RoboDK station: kr30 cnc 101019 2.rdk

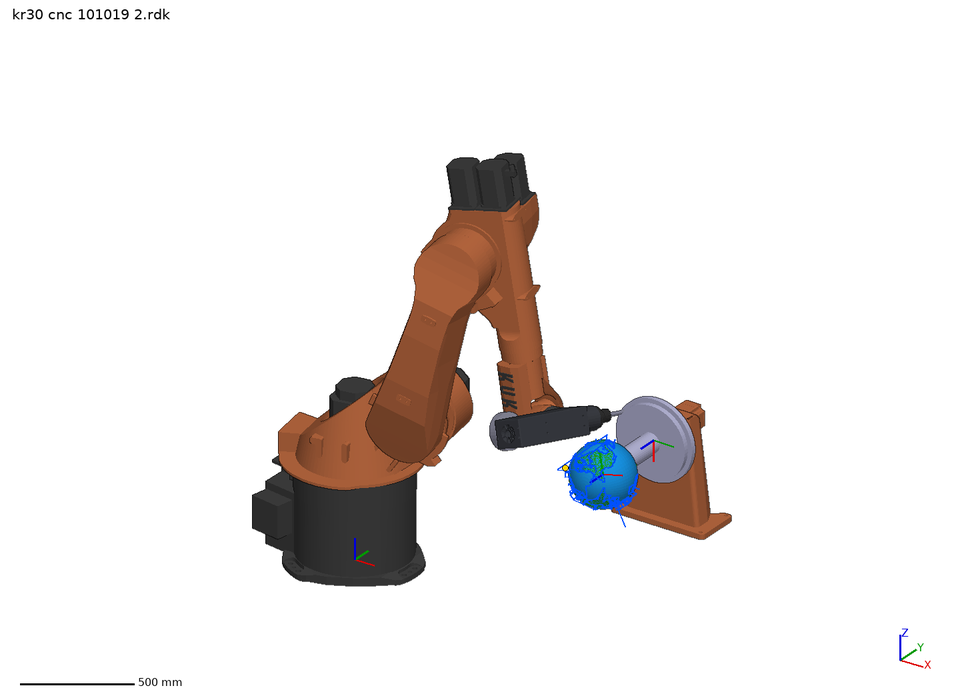
[picture v0: the station drawn from its stored meshes, robots at their saved joint values, targets as dots, program paths as lines]
Station kr30 cnc 101019 2. Poses are relative to the parent item; angles as X-Y-Z fixed-axis rotations.
  - frame KUKA KR 30 HA Base at (0, 0, 0) mm
    - robot KUKA KR 30 HA: 6 axes, payload 30 kg, reach 2033 mm, repeatability 0.05 mm, weight 665 kg
        modified DH rows (alpha deg, a mm, theta deg, d mm): 0, 0, 0, 815; -90, 350, 0, 0; 0, 850, -90, 0; -90, 145, 0, 820; 90, 0, 0, 0; -90, 0, 180, 170
        joint limits [-185, -135, -120, -350, -119, -350] to [185, 35, 158, 350, 119, 350]; home [0, -90, 90, 0, 0, 0]; saved at [-9.82, -73.833, 154.586, -18.357, -102.464, -76.723]
      - tool Spindle, TCP at (249.17, -0.03, 160.93) mm, rotated rx 0 ry 90 rz 0 deg, size 170 x 692.9 x 256 mm
  - frame KUKA KP1 MD250 Base at (1360.87, 339.35, 824.43) mm, rotated rx -93.1 ry 88.62 rz 178.42 deg
    - robot KUKA KP1 MD250: 1 axes, payload 250 kg
        modified DH rows (alpha deg, a mm, theta deg, d mm): 0, 0, 0, 0
        joint limits [-180] to [180]; home [0]; saved at [-257.733]
      - frame MillingEarth at (0, 0, 402.47) mm
        - object Earth at (0, 0, 0) mm, size 359.7 x 359.7 x 550 mm
  - machining project MillingEarth Settings: C:/Users/albert/Desktop/RoboDK/Deploy/RoboDK_vc2013x64/Library/Milling Earth (5axis).nc | rotZ(0) | rotX(0)*rotY(0) | rotZ(90)
  - program MillingEarth (2694 instructions, listed below)
  - program Prog2 (0 instructions, listed below)
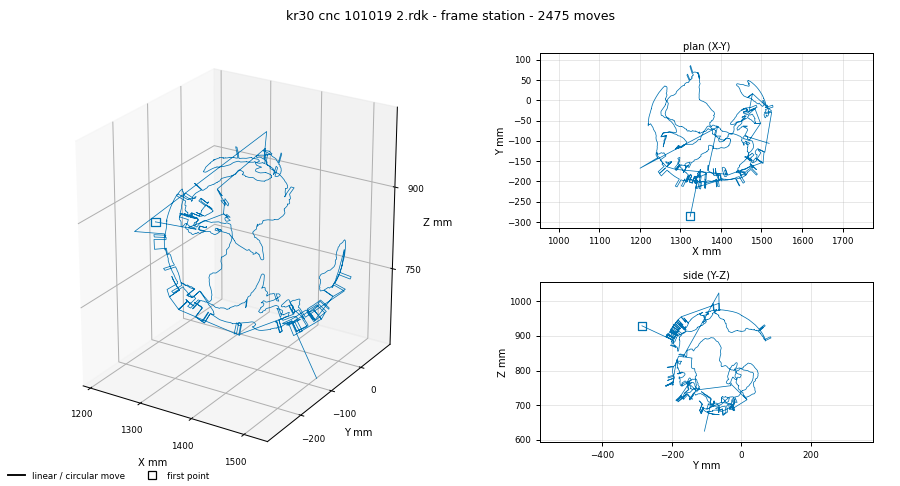
[picture p0: tool path of kr30 cnc 101019 2.rdk in frame station, 2475 of 2475 moves have a stored position in this frame; points joined in program order, loops and branches not executed]

--- program MillingEarth (robot KUKA KR 30 HA) ---
  Call onMillingEarth_Start
  Set Ref.: MillingEarth
  Set Tool: Spindle
  Show Spindle
  Set speed (16.7 mm/s)
  Call SetCLW
  Call SetRPM(70.0)
  Set speed (1000.0 mm/s)
  MoveJ 1 to (-32.4, 113.46, 221.55) mm, rotated rx -152.37 ry 0 rz -164.91 deg; joints [17.149, -48.365, 79.155, 0, 59.444, -43.7, -13.927]
  MoveL 2 to (-32.4, 113.46, 221.55) mm, rotated rx -152.37 ry 0 rz -164.91 deg; joints [17.149, -48.365, 79.155, 0, 59.444, -43.7, -13.926]
  Call onMillingEarth_Approach
  MoveL 3 to (-20.33, 68.69, 132.95) mm, rotated rx -152.37 ry 0 rz -164.91 deg; joints [14.531, -51.571, 85.433, 1.012, 59.444, -46.856, -17.119]
  Call onMillingEarth_PathStart
  MoveL 4 to (-20.33, 68.69, 132.95) mm, rotated rx -152.37 ry 0 rz -164.91 deg; joints [14.531, -51.571, 85.433, 1.012, 59.444, -46.856, -17.119]
  MoveL 5 to (-19.96, 69.22, 132.73) mm, rotated rx -152.2 ry 0 rz -165.3 deg; joints [14.503, -51.529, 85.357, 0.999, 59.444, -46.702, -16.7]
  Set speed (16.7 mm/s)
  MoveL 6 to (-22.33, 78.24, 150.42) mm, rotated rx -152.2 ry 0 rz -165.3 deg; joints [15.035, -50.886, 84.143, 0.841, 59.444, -46.082, -16.114]
  Set speed (1000.0 mm/s)
  MoveL 7 to (39.62, 97.38, 134.89) mm, rotated rx -142.85 ry 0 rz 157.38 deg; joints [13.369, -48.767, 80.092, 0.147, 59.444, -38.037, 23.226]
  Set speed (5.0 mm/s)
  MoveL 8 to (34.97, 86.23, 118.95) mm, rotated rx -142.85 ry 0 rz 157.38 deg; joints [12.91, -49.457, 81.504, 0.356, 59.444, -38.604, 22.481]
  Set speed (16.7 mm/s)
  MoveL 9 to (35.17, 86.21, 118.9) mm, rotated rx -142.83 ry 0 rz 157.26 deg; joints [12.906, -49.452, 81.493, 0.354, 59.444, -38.581, 22.605]
  MoveL 10 to (35.37, 86.18, 118.87) mm, rotated rx -142.83 ry 0 rz 157.26 deg; joints [12.904, -49.443, 81.493, 0.355, 59.439, -38.583, 22.602]
  MoveL 11 to (39.2, 85.43, 118.2) mm, rotated rx -142.42 ry 0 rz 154.93 deg; joints [12.831, -49.365, 81.337, 0.33, 59.439, -38.237, 25.012]
  MoveL 12 to (44.37, 96.48, 134.05) mm, rotated rx -142.42 ry 0 rz 154.93 deg; joints [13.286, -48.674, 79.917, 0.119, 59.439, -37.672, 25.764]
  Set speed (1000.0 mm/s)
  MoveL 13 to (45.45, 92.09, 136.75) mm, rotated rx -142.45 ry 0 rz 154.62 deg; joints [13.396, -48.674, 80.171, 0.201, 59.442, -37.638, 25.808]
  Set speed (5.0 mm/s)
  MoveL 14 to (40.23, 81.08, 120.9) mm, rotated rx -142.45 ry 0 rz 154.62 deg; joints [12.942, -49.369, 81.594, 0.41, 59.443, -38.201, 25.058]
  Set speed (16.7 mm/s)
  MoveL 15 to (37.93, 80.72, 121.87) mm, rotated rx -143.08 ry 0 rz 155.86 deg; joints [13.052, -49.49, 81.836, 0.45, 59.443, -38.738, 23.689]
  MoveL 16 to (37.59, 80.7, 121.99) mm, rotated rx -143.15 ry 0 rz 156.04 deg; joints [13.065, -49.505, 81.863, 0.454, 59.443, -38.795, 23.499]
  MoveL 17 to (35.64, 80.36, 122.8) mm, rotated rx -143.67 ry 0 rz 157.12 deg; joints [13.157, -49.609, 82.069, 0.489, 59.443, -39.247, 22.314]
  MoveL 18 to (35.2, 80.32, 122.95) mm, rotated rx -143.67 ry 0 rz 157.12 deg; joints [13.164, -49.63, 82.075, 0.489, 59.457, -39.24, 22.314]
  MoveL 19 to (34.17, 80.49, 123.13) mm, rotated rx -143.67 ry 0 rz 157.12 deg; joints [13.173, -49.678, 82.075, 0.482, 59.484, -39.227, 22.337]
  MoveL 20 to (33.97, 80.56, 123.14) mm, rotated rx -143.68 ry 0 rz 157.26 deg; joints [13.174, -49.679, 82.077, 0.483, 59.484, -39.233, 22.196]
  MoveL 21 to (33.46, 80.79, 123.13) mm, rotated rx -143.68 ry 0 rz 157.26 deg; joints [13.175, -49.708, 82.074, 0.473, 59.484, -39.227, 22.228]
  MoveL 22 to (32.55, 81.6, 122.84) mm, rotated rx -143.68 ry 0 rz 157.26 deg; joints [13.166, -49.754, 82.043, 0.449, 59.484, -39.223, 22.308]
  MoveL 23 to (31.58, 82.93, 122.2) mm, rotated rx -143.26 ry 0 rz 158.18 deg; joints [13.092, -49.671, 81.88, 0.422, 59.484, -38.865, 21.471]
  MoveL 24 to (31.06, 83.97, 121.62) mm, rotated rx -143.25 ry 0 rz 158.2 deg; joints [13.068, -49.685, 81.82, 0.399, 59.484, -38.861, 21.523]
  MoveL 25 to (31.07, 84.77, 121.06) mm, rotated rx -143.23 ry 0 rz 158.22 deg; joints [13.044, -49.671, 81.765, 0.386, 59.483, -38.866, 21.548]
  MoveL 26 to (31.31, 85.29, 120.63) mm, rotated rx -143.22 ry 0 rz 158.24 deg; joints [13.025, -49.647, 81.723, 0.38, 59.483, -38.874, 21.553]
  MoveL 27 to (31.95, 85.85, 120.07) mm, rotated rx -143.21 ry 0 rz 158.26 deg; joints [12.999, -49.604, 81.676, 0.373, 59.469, -38.883, 21.553]
  MoveL 28 to (32.84, 86.09, 119.65) mm, rotated rx -143.2 ry 0 rz 158.27 deg; joints [12.98, -49.563, 81.657, 0.367, 59.428, -38.887, 21.553]
  MoveL 29 to (34.47, 86.24, 119.09) mm, rotated rx -142.85 ry 0 rz 157.38 deg; joints [12.918, -49.496, 81.523, 0.345, 59.428, -38.591, 22.517]
  MoveL 30 to (39.12, 97.38, 135.03) mm, rotated rx -142.85 ry 0 rz 157.38 deg; joints [13.377, -48.806, 80.112, 0.137, 59.428, -38.024, 23.262]
  Set speed (1000.0 mm/s)
  MoveL 31 to (36.17, 117.37, 119.01) mm, rotated rx -134.2 ry 0 rz 164.03 deg; joints [11.734, -47.132, 76.943, -0.298, 59.428, -30.795, 18.15]
  Set speed (5.0 mm/s)
  MoveL 32 to (32.22, 103.58, 105.07) mm, rotated rx -134.2 ry 0 rz 164.03 deg; joints [11.348, -47.847, 78.519, -0.063, 59.428, -31.299, 17.264]
  Set speed (16.7 mm/s)
  MoveL 33 to (31.89, 100.84, 107.81) mm, rotated rx -135.66 ry 0 rz 163.8 deg; joints [11.629, -48.075, 79.013, 0.01, 59.428, -32.518, 17.226]
  MoveL 34 to (35.79, 114.26, 122.11) mm, rotated rx -135.66 ry 0 rz 163.8 deg; joints [12.027, -47.363, 77.462, -0.222, 59.428, -32.002, 18.089]
  Set speed (1000.0 mm/s)
  MoveL 35 to (30.39, 115.24, 122.66) mm, rotated rx -135.75 ry 0 rz 164.03 deg; joints [12.066, -47.602, 77.462, -0.26, 59.533, -32.027, 17.992]
  Set speed (5.0 mm/s)
  MoveL 36 to (26.55, 101.82, 108.33) mm, rotated rx -135.75 ry 0 rz 164.03 deg; joints [11.666, -48.313, 79.006, -0.028, 59.533, -32.543, 17.134]
  Set speed (16.7 mm/s)
  MoveL 37 to (26.92, 104.59, 105.56) mm, rotated rx -134.26 ry 0 rz 164.25 deg; joints [11.381, -48.081, 78.504, -0.101, 59.533, -31.302, 17.192]
  MoveL 38 to (30.8, 118.38, 119.52) mm, rotated rx -134.26 ry 0 rz 164.25 deg; joints [11.768, -47.367, 76.934, -0.336, 59.533, -30.798, 18.073]
  Set speed (1000.0 mm/s)
  MoveL 39 to (18.54, 129.47, 110.19) mm, rotated rx -130.91 ry 0 rz 171.49 deg; joints [11.006, -46.736, 75.687, -0.48, 59.533, -28.141, 11.458]
  Set speed (5.0 mm/s)
  MoveL 40 to (16.3, 114.52, 97.09) mm, rotated rx -130.91 ry 0 rz 171.49 deg; joints [10.647, -47.452, 77.314, -0.24, 59.533, -28.616, 10.522]
  Set speed (16.7 mm/s)
  MoveL 41 to (17.17, 114.58, 96.87) mm, rotated rx -130.8 ry 0 rz 171.07 deg; joints [10.625, -47.437, 77.281, -0.245, 59.533, -28.526, 10.961]
  MoveL 42 to (17.11, 114.6, 96.86) mm, rotated rx -128.95 ry 0 rz 171.63 deg; joints [10.392, -47.226, 76.933, -0.275, 59.533, -26.899, 10.541]
  MoveL 43 to (16.23, 114.67, 96.93) mm, rotated rx -128.98 ry 0 rz 172.06 deg; joints [10.399, -47.23, 76.942, -0.273, 59.535, -26.926, 10.101]
  MoveL 44 to (18.38, 130.06, 109.51) mm, rotated rx -128.98 ry 0 rz 172.06 deg; joints [10.74, -46.507, 75.283, -0.515, 59.535, -26.468, 11.062]
  Set speed (1000.0 mm/s)
  MoveL 45 to (51.72, 163.01, 1.41) mm, rotated rx -91.23 ry 0 rz 162.75 deg; joints [1.995, -46.507, 71.751, -0.724, 56.15, 2.635, 27.263]
  Set speed (5.0 mm/s)
  MoveL 46 to (45.79, 143.91, 0.98) mm, rotated rx -91.23 ry 0 rz 162.75 deg; joints [2.004, -47.144, 73.595, -0.637, 56.154, 2.607, 26.05]
  Set speed (16.7 mm/s)
  MoveL 47 to (46.25, 143.76, 1.2) mm, rotated rx -91.32 ry 0 rz 162.56 deg; joints [2.023, -47.144, 73.594, -0.64, 56.152, 2.544, 26.237]
  MoveL 48 to (46.82, 143.57, 1.59) mm, rotated rx -91.32 ry 0 rz 162.56 deg; joints [2.036, -47.115, 73.594, -0.641, 56.139, 2.557, 26.221]
  MoveL 49 to (49.93, 142.45, 4.46) mm, rotated rx -92.41 ry 0 rz 161.31 deg; joints [2.289, -47.115, 73.581, -0.683, 56.12, 1.741, 27.508]
  MoveL 50 to (49.93, 142.46, 4.45) mm, rotated rx -92.58 ry 0 rz 161.02 deg; joints [2.313, -47.154, 73.581, -0.689, 56.13, 1.6, 27.828]
  MoveL 51 to (53.02, 141.29, 5.69) mm, rotated rx -93.05 ry 0 rz 159.77 deg; joints [2.422, -47.154, 73.578, -0.707, 56.124, 1.249, 29.091]
  MoveL 52 to (53.52, 141.09, 5.97) mm, rotated rx -93.05 ry 0 rz 159.77 deg; joints [2.431, -47.127, 73.578, -0.707, 56.114, 1.258, 29.075]
  MoveL 53 to (54.32, 140.74, 7.02) mm, rotated rx -93.05 ry 0 rz 159.77 deg; joints [2.465, -47.084, 73.578, -0.71, 56.096, 1.295, 29.051]
  MoveL 54 to (54.41, 140.69, 7.24) mm, rotated rx -93.13 ry 0 rz 159.73 deg; joints [2.484, -47.084, 73.578, -0.714, 56.095, 1.233, 29.088]
  MoveL 55 to (54.58, 140.57, 8.16) mm, rotated rx -93.13 ry 0 rz 159.73 deg; joints [2.515, -47.074, 73.578, -0.718, 56.089, 1.266, 29.085]
  MoveL 56 to (54.59, 140.48, 9.51) mm, rotated rx -93.64 ry 0 rz 159.71 deg; joints [2.634, -47.074, 73.577, -0.737, 56.085, 0.883, 29.106]
  MoveL 57 to (54.58, 140.49, 9.48) mm, rotated rx -94.31 ry 0 rz 159.4 deg; joints [2.73, -47.115, 73.577, -0.754, 56.097, 0.318, 29.449]
  MoveL 58 to (58.8, 138.43, 13.63) mm, rotated rx -95.89 ry 0 rz 157.62 deg; joints [3.095, -47.113, 73.586, -0.811, 56.097, -0.865, 31.221]
  MoveL 59 to (58.75, 138.46, 13.59) mm, rotated rx -96.1 ry 0 rz 157.16 deg; joints [3.126, -47.174, 73.586, -0.819, 56.123, -1.045, 31.719]
  MoveL 60 to (63.19, 136.41, 14.38) mm, rotated rx -96.4 ry 0 rz 155.3 deg; joints [3.195, -47.174, 73.59, -0.829, 56.123, -1.269, 33.577]
  MoveL 61 to (63.44, 136.29, 14.44) mm, rotated rx -96.4 ry 0 rz 155.3 deg; joints [3.197, -47.16, 73.59, -0.829, 56.119, -1.268, 33.568]
  MoveL 62 to (63.67, 136.17, 14.51) mm, rotated rx -96.43 ry 0 rz 155.2 deg; joints [3.203, -47.16, 73.59, -0.83, 56.119, -1.288, 33.667]
  MoveL 63 to (65.41, 135.28, 15.07) mm, rotated rx -96.66 ry 0 rz 154.35 deg; joints [3.257, -47.171, 73.59, -0.838, 56.13, -1.47, 34.516]
  MoveL 64 to (65.72, 135.13, 15.13) mm, rotated rx -96.69 ry 0 rz 154.22 deg; joints [3.261, -47.171, 73.591, -0.839, 56.13, -1.485, 34.646]
  MoveL 65 to (68.28, 133.79, 15.64) mm, rotated rx -96.88 ry 0 rz 153.13 deg; joints [3.306, -47.169, 73.594, -0.845, 56.13, -1.63, 35.729]
  MoveL 66 to (68.86, 133.47, 15.86) mm, rotated rx -96.88 ry 0 rz 153.13 deg; joints [3.313, -47.135, 73.594, -0.844, 56.119, -1.624, 35.707]
  MoveL 67 to (69.74, 132.95, 16.36) mm, rotated rx -97.07 ry 0 rz 152.75 deg; joints [3.357, -47.133, 73.595, -0.85, 56.125, -1.766, 36.083]
  MoveL 68 to (69.89, 132.86, 16.45) mm, rotated rx -97.07 ry 0 rz 152.75 deg; joints [3.36, -47.124, 73.595, -0.85, 56.122, -1.763, 36.077]
  MoveL 69 to (76.53, 128.45, 21.19) mm, rotated rx -98.88 ry 0 rz 149.71 deg; joints [3.778, -47.124, 73.638, -0.908, 56.143, -3.127, 39.054]
  MoveL 70 to (76.49, 128.48, 21.19) mm, rotated rx -98.98 ry 0 rz 148.97 deg; joints [3.794, -47.219, 73.638, -0.916, 56.183, -3.206, 39.853]
  MoveL 71 to (80.12, 126.44, 20.02) mm, rotated rx -98.53 ry 0 rz 147.38 deg; joints [3.69, -47.219, 73.625, -0.902, 56.176, -2.867, 41.464]
  MoveL 72 to (80.83, 126, 19.93) mm, rotated rx -98.53 ry 0 rz 147.38 deg; joints [3.686, -47.179, 73.625, -0.899, 56.16, -2.872, 41.439]
  MoveL 73 to (81.28, 125.71, 19.96) mm, rotated rx -98.54 ry 0 rz 147.17 deg; joints [3.689, -47.179, 73.625, -0.9, 56.16, -2.881, 41.642]
  MoveL 74 to (81.75, 125.39, 20.06) mm, rotated rx -98.54 ry 0 rz 147.17 deg; joints [3.692, -47.15, 73.625, -0.898, 56.15, -2.879, 41.623]
  MoveL 75 to (86.58, 121.8, 21.83) mm, rotated rx -99.22 ry 0 rz 144.87 deg; joints [3.849, -47.15, 73.644, -0.919, 56.161, -3.392, 43.899]
  MoveL 76 to (87.18, 121.32, 22.1) mm, rotated rx -99.31 ry 0 rz 144.62 deg; joints [3.87, -47.145, 73.647, -0.921, 56.161, -3.457, 44.142]
  MoveL 77 to (91.51, 117.76, 23.78) mm, rotated rx -99.97 ry 0 rz 142.43 deg; joints [4.02, -47.145, 73.663, -0.94, 56.184, -3.955, 46.29]
  MoveL 78 to (91.73, 117.56, 23.89) mm, rotated rx -99.97 ry 0 rz 142.43 deg; joints [4.023, -47.13, 73.664, -0.939, 56.179, -3.952, 46.28]
  MoveL 79 to (92.05, 117.28, 24.08) mm, rotated rx -100.04 ry 0 rz 142.27 deg; joints [4.04, -47.13, 73.667, -0.942, 56.18, -4.006, 46.437]
  MoveL 80 to (92.22, 117.12, 24.19) mm, rotated rx -100.04 ry 0 rz 142.27 deg; joints [4.044, -47.118, 73.666, -0.941, 56.178, -4.003, 46.428]
  MoveL 81 to (94.43, 114.96, 25.97) mm, rotated rx -100.72 ry 0 rz 141.09 deg; joints [4.2, -47.118, 73.692, -0.96, 56.194, -4.518, 47.571]
  MoveL 82 to (96.38, 113.21, 26.49) mm, rotated rx -101.03 ry 0 rz 139.79 deg; joints [4.263, -47.144, 73.692, -0.968, 56.231, -4.763, 48.857]
  MoveL 83 to (96.7, 112.9, 26.63) mm, rotated rx -101.03 ry 0 rz 139.79 deg; joints [4.267, -47.121, 73.692, -0.967, 56.225, -4.759, 48.84]
  MoveL 84 to (96.94, 112.66, 26.77) mm, rotated rx -101.08 ry 0 rz 139.66 deg; joints [4.279, -47.121, 73.694, -0.968, 56.226, -4.8, 48.967]
  MoveL 85 to (97.15, 112.45, 26.91) mm, rotated rx -101.08 ry 0 rz 139.66 deg; joints [4.284, -47.105, 73.694, -0.967, 56.223, -4.796, 48.955]
  MoveL 86 to (99.43, 109.95, 28.85) mm, rotated rx -101.83 ry 0 rz 138.37 deg; joints [4.455, -47.105, 73.726, -0.986, 56.245, -5.361, 50.196]
  MoveL 87 to (99.68, 109.66, 29.07) mm, rotated rx -101.92 ry 0 rz 138.21 deg; joints [4.475, -47.105, 73.73, -0.988, 56.249, -5.428, 50.343]
  MoveL 88 to (100.05, 109.21, 29.52) mm, rotated rx -101.92 ry 0 rz 138.21 deg; joints [4.489, -47.074, 73.73, -0.987, 56.246, -5.415, 50.314]
  MoveL 89 to (101.45, 107.18, 32.04) mm, rotated rx -102.89 ry 0 rz 137.28 deg; joints [4.712, -47.075, 73.778, -1.01, 56.278, -6.156, 51.167]
  MoveL 90 to (101.64, 106.86, 32.53) mm, rotated rx -102.89 ry 0 rz 137.28 deg; joints [4.728, -47.055, 73.779, -1.009, 56.278, -6.14, 51.146]
  MoveL 91 to (101.66, 106.43, 33.85) mm, rotated rx -102.89 ry 0 rz 137.28 deg; joints [4.772, -47.041, 73.791, -1.013, 56.278, -6.094, 51.121]
  MoveL 92 to (101.59, 106.39, 34.17) mm, rotated rx -103.02 ry 0 rz 137.29 deg; joints [4.8, -47.041, 73.798, -1.015, 56.283, -6.188, 51.102]
  MoveL 93 to (101.26, 106.41, 35.09) mm, rotated rx -103.02 ry 0 rz 137.29 deg; joints [4.831, -47.047, 73.798, -1.017, 56.305, -6.156, 51.086]
  MoveL 94 to (100.18, 106.74, 37.1) mm, rotated rx -103.8 ry 0 rz 137.69 deg; joints [5.01, -47.047, 73.842, -1.033, 56.338, -6.756, 50.61]
  MoveL 95 to (100.18, 106.75, 37.07) mm, rotated rx -104.74 ry 0 rz 137.63 deg; joints [5.141, -47.047, 73.868, -1.042, 56.38, -7.555, 50.606]
  MoveL 96 to (101.87, 103.05, 42.54) mm, rotated rx -107.02 ry 0 rz 136.04 deg; joints [5.645, -47.047, 74.005, -1.07, 56.529, -9.322, 51.922]
  MoveL 97 to (102.05, 102.73, 42.88) mm, rotated rx -107.16 ry 0 rz 135.9 deg; joints [5.676, -47.047, 74.015, -1.072, 56.537, -9.425, 52.043]
  MoveL 98 to (104.05, 99.2, 46.26) mm, rotated rx -108.54 ry 0 rz 134.31 deg; joints [5.982, -47.047, 74.116, -1.081, 56.635, -10.493, 53.437]
  MoveL 99 to (104.28, 98.54, 47.15) mm, rotated rx -108.59 ry 0 rz 134.31 deg; joints [6.018, -47.015, 74.131, -1.079, 56.635, -10.506, 53.387]
  MoveL 100 to (104.13, 98.18, 48.22) mm, rotated rx -108.63 ry 0 rz 134.31 deg; joints [6.06, -47.013, 74.153, -1.081, 56.635, -10.509, 53.359]
  MoveL 101 to (103.98, 98.01, 48.88) mm, rotated rx -108.9 ry 0 rz 134.31 deg; joints [6.119, -47.013, 74.176, -1.082, 56.654, -10.716, 53.322]
  MoveL 102 to (103.97, 98.04, 48.86) mm, rotated rx -109.5 ry 0 rz 134.07 deg; joints [6.202, -47.014, 74.176, -1.077, 56.743, -11.239, 53.472]
  MoveL 103 to (104.32, 97.19, 49.77) mm, rotated rx -109.87 ry 0 rz 133.73 deg; joints [6.284, -47.014, 74.209, -1.077, 56.771, -11.525, 53.754]
  MoveL 104 to (104.27, 97.22, 49.84) mm, rotated rx -109.04 ry 0 rz 132.02 deg; joints [6.179, -47.246, 74.182, -1.106, 56.771, -10.79, 55.725]
  MoveL 105 to (104.53, 98.86, 45.91) mm, rotated rx -107.47 ry 0 rz 132.44 deg; joints [5.826, -47.246, 74.054, -1.096, 56.663, -9.572, 55.539]
  MoveL 106 to (104.48, 99.07, 45.58) mm, rotated rx -107.19 ry 0 rz 132.57 deg; joints [5.777, -47.246, 74.044, -1.095, 56.636, -9.348, 55.449]
  MoveL 107 to (104.22, 100.62, 42.67) mm, rotated rx -106.04 ry 0 rz 133.09 deg; joints [5.517, -47.246, 73.959, -1.082, 56.568, -8.458, 55.076]
  MoveL 108 to (118.26, 113.75, 48.19) mm, rotated rx -106.04 ry 0 rz 133.09 deg; joints [5.653, -46.589, 72.136, -1.276, 56.567, -8.236, 56.255]
  Set speed (1000.0 mm/s)
  MoveL 109 to (121.75, 111.27, 45.2) mm, rotated rx -106.02 ry 0 rz 132.91 deg; joints [5.547, -46.443, 72.136, -1.261, 56.421, -8.333, 56.435]
  Set speed (5.0 mm/s)
  MoveL 110 to (107.67, 98.18, 39.68) mm, rotated rx -106.02 ry 0 rz 132.91 deg; joints [5.411, -47.099, 73.963, -1.068, 56.421, -8.555, 55.251]
  Set speed (16.7 mm/s)
  MoveL 111 to (109.17, 95.75, 41.47) mm, rotated rx -106.73 ry 0 rz 131.8 deg; joints [5.57, -47.099, 74.013, -1.077, 56.46, -9.097, 56.269]
  MoveL 112 to (109.28, 95.57, 41.61) mm, rotated rx -106.78 ry 0 rz 131.72 deg; joints [5.582, -47.099, 74.017, -1.078, 56.463, -9.138, 56.345]
  MoveL 113 to (110.67, 92.99, 43.73) mm, rotated rx -107.58 ry 0 rz 130.65 deg; joints [5.765, -47.099, 74.085, -1.088, 56.497, -9.747, 57.313]
  MoveL 114 to (110.84, 92.61, 44.1) mm, rotated rx -107.58 ry 0 rz 130.65 deg; joints [5.777, -47.078, 74.087, -1.086, 56.497, -9.736, 57.289]
  MoveL 115 to (110.92, 91.99, 45.19) mm, rotated rx -107.58 ry 0 rz 130.65 deg; joints [5.813, -47.053, 74.101, -1.085, 56.497, -9.701, 57.251]
  MoveL 116 to (110.89, 91.91, 45.44) mm, rotated rx -107.68 ry 0 rz 130.63 deg; joints [5.835, -47.053, 74.109, -1.086, 56.504, -9.776, 57.255]
  MoveL 117 to (110.71, 91.74, 46.19) mm, rotated rx -107.68 ry 0 rz 130.63 deg; joints [5.86, -47.053, 74.118, -1.087, 56.51, -9.75, 57.24]
  MoveL 118 to (110.22, 91.6, 47.62) mm, rotated rx -108.25 ry 0 rz 130.72 deg; joints [5.989, -47.053, 74.165, -1.09, 56.548, -10.194, 57.07]
  MoveL 119 to (110.22, 91.62, 47.57) mm, rotated rx -109.14 ry 0 rz 130.3 deg; joints [6.11, -47.061, 74.165, -1.086, 56.679, -10.967, 57.364]
  MoveL 120 to (112.14, 87.75, 50.32) mm, rotated rx -110.24 ry 0 rz 128.62 deg; joints [6.355, -47.061, 74.261, -1.088, 56.761, -11.82, 58.874]
  MoveL 121 to (112.4, 86.84, 51.32) mm, rotated rx -110.24 ry 0 rz 128.62 deg; joints [6.388, -47.017, 74.274, -1.082, 56.761, -11.79, 58.816]
  MoveL 122 to (112.13, 86.41, 52.6) mm, rotated rx -110.24 ry 0 rz 128.62 deg; joints [6.431, -47.016, 74.3, -1.083, 56.761, -11.746, 58.79]
  MoveL 123 to (112.01, 86.37, 52.93) mm, rotated rx -110.38 ry 0 rz 128.64 deg; joints [6.461, -47.017, 74.313, -1.083, 56.77, -11.85, 58.747]
  MoveL 124 to (111.32, 86.54, 54.09) mm, rotated rx -110.38 ry 0 rz 128.64 deg; joints [6.5, -47.029, 74.313, -1.081, 56.82, -11.812, 58.709]
  MoveL 125 to (110.56, 86.95, 54.96) mm, rotated rx -110.73 ry 0 rz 128.96 deg; joints [6.579, -47.033, 74.352, -1.081, 56.843, -12.09, 58.33]
  MoveL 126 to (110.59, 86.95, 54.91) mm, rotated rx -111.91 ry 0 rz 128.97 deg; joints [6.74, -47.043, 74.434, -1.081, 56.887, -13.111, 58.207]
  MoveL 127 to (110.98, 85.3, 56.68) mm, rotated rx -112.64 ry 0 rz 128.35 deg; joints [6.9, -47.06, 74.524, -1.081, 56.923, -13.674, 58.722]
  MoveL 128 to (111.01, 84.82, 57.35) mm, rotated rx -112.64 ry 0 rz 128.35 deg; joints [6.922, -47.042, 74.537, -1.078, 56.923, -13.653, 58.691]
  MoveL 129 to (110.99, 84.64, 57.66) mm, rotated rx -112.76 ry 0 rz 128.3 deg; joints [6.95, -47.046, 74.554, -1.078, 56.929, -13.752, 58.721]
  MoveL 130 to (110.91, 84.43, 58.11) mm, rotated rx -112.76 ry 0 rz 128.3 deg; joints [6.965, -47.043, 74.565, -1.077, 56.929, -13.737, 58.708]
  MoveL 131 to (110.03, 83.05, 61.67) mm, rotated rx -114.23 ry 0 rz 128.08 deg; joints [7.289, -47.102, 74.782, -1.077, 56.976, -14.882, 58.727]
  MoveL 132 to (109.88, 82.87, 62.17) mm, rotated rx -114.4 ry 0 rz 128.06 deg; joints [7.328, -47.111, 74.811, -1.077, 56.98, -15.003, 58.718]
  MoveL 133 to (109.06, 81.95, 64.77) mm, rotated rx -115.48 ry 0 rz 127.97 deg; joints [7.566, -47.171, 74.996, -1.077, 56.996, -15.847, 58.674]
  MoveL 134 to (109.07, 81.98, 64.73) mm, rotated rx -116.1 ry 0 rz 127.61 deg; joints [7.65, -47.221, 75.046, -1.077, 57.042, -16.387, 58.982]
  MoveL 135 to (109.68, 79.86, 66.33) mm, rotated rx -116.77 ry 0 rz 126.75 deg; joints [7.796, -47.266, 75.171, -1.077, 57.044, -16.909, 59.764]
  MoveL 136 to (109.69, 79.87, 66.3) mm, rotated rx -116.91 ry 0 rz 126.48 deg; joints [7.815, -47.29, 75.173, -1.077, 57.075, -17.033, 60.026]
  MoveL 137 to (110.88, 77.27, 67.41) mm, rotated rx -117.38 ry 0 rz 125.3 deg; joints [7.916, -47.323, 75.264, -1.077, 57.075, -17.396, 61.148]
  MoveL 138 to (111.03, 76.87, 67.61) mm, rotated rx -117.38 ry 0 rz 125.3 deg; joints [7.922, -47.301, 75.267, -1.072, 57.075, -17.392, 61.123]
  MoveL 139 to (111.15, 76.07, 68.3) mm, rotated rx -117.38 ry 0 rz 125.3 deg; joints [7.945, -47.267, 75.284, -1.065, 57.075, -17.373, 61.072]
  MoveL 140 to (111.14, 75.85, 68.56) mm, rotated rx -117.49 ry 0 rz 125.23 deg; joints [7.969, -47.275, 75.306, -1.064, 57.075, -17.459, 61.131]
  MoveL 141 to (111.07, 75.48, 69.1) mm, rotated rx -117.49 ry 0 rz 125.23 deg; joints [7.987, -47.267, 75.322, -1.062, 57.075, -17.442, 61.107]
  MoveL 142 to (110.3, 73.8, 72.07) mm, rotated rx -118.76 ry 0 rz 124.83 deg; joints [8.263, -47.364, 75.582, -1.057, 57.075, -18.44, 61.346]
  MoveL 143 to (110.19, 73.63, 72.41) mm, rotated rx -118.76 ry 0 rz 124.83 deg; joints [8.275, -47.364, 75.593, -1.056, 57.076, -18.429, 61.335]
  MoveL 144 to (110.02, 73.45, 72.86) mm, rotated rx -118.95 ry 0 rz 124.8 deg; joints [8.317, -47.379, 75.634, -1.055, 57.076, -18.581, 61.334]
  MoveL 145 to (109.94, 73.37, 73.05) mm, rotated rx -118.95 ry 0 rz 124.8 deg; joints [8.323, -47.38, 75.64, -1.054, 57.078, -18.575, 61.327]
  MoveL 146 to (108.02, 71.92, 77.24) mm, rotated rx -120.78 ry 0 rz 124.76 deg; joints [8.716, -47.532, 76.041, -1.04, 57.078, -20.017, 61.124]
  MoveL 147 to (107.85, 71.77, 77.62) mm, rotated rx -120.99 ry 0 rz 124.74 deg; joints [8.757, -47.549, 76.084, -1.038, 57.078, -20.182, 61.112]
  MoveL 148 to (105.63, 70.25, 81.94) mm, rotated rx -122.86 ry 0 rz 124.76 deg; joints [9.159, -47.722, 76.531, -1.015, 57.078, -21.661, 60.826]
  MoveL 149 to (104.84, 70.16, 83.03) mm, rotated rx -122.86 ry 0 rz 124.76 deg; joints [9.198, -47.757, 76.574, -1.015, 57.085, -21.621, 60.81]
  MoveL 150 to (104.53, 70.23, 83.36) mm, rotated rx -123.01 ry 0 rz 124.87 deg; joints [9.229, -47.771, 76.61, -1.013, 57.085, -21.738, 60.68]
  MoveL 151 to (104.24, 70.33, 83.64) mm, rotated rx -123.01 ry 0 rz 124.87 deg; joints [9.24, -47.785, 76.618, -1.013, 57.094, -21.728, 60.677]
  MoveL 152 to (101.64, 71.39, 85.9) mm, rotated rx -124.05 ry 0 rz 125.95 deg; joints [9.458, -47.887, 76.878, -0.995, 57.094, -22.56, 59.432]
  MoveL 153 to (101.65, 71.39, 85.9) mm, rotated rx -124.25 ry 0 rz 126.11 deg; joints [9.483, -47.88, 76.907, -0.989, 57.095, -22.736, 59.237]
  MoveL 154 to (99.95, 71.26, 87.98) mm, rotated rx -125.31 ry 0 rz 126.59 deg; joints [9.696, -47.979, 77.172, -0.968, 57.095, -23.594, 58.597]
  MoveL 155 to (99.56, 71.29, 88.39) mm, rotated rx -125.31 ry 0 rz 126.59 deg; joints [9.712, -47.997, 77.189, -0.968, 57.102, -23.579, 58.592]
  MoveL 156 to (99.1, 71.39, 88.83) mm, rotated rx -125.52 ry 0 rz 126.75 deg; joints [9.755, -48.019, 77.243, -0.964, 57.102, -23.745, 58.394]
  MoveL 157 to (98.75, 71.49, 89.13) mm, rotated rx -125.52 ry 0 rz 126.75 deg; joints [9.766, -48.036, 77.253, -0.963, 57.112, -23.734, 58.39]
  MoveL 158 to (93.79, 73.31, 92.93) mm, rotated rx -127.33 ry 0 rz 128.89 deg; joints [10.139, -48.235, 77.746, -0.921, 57.112, -25.196, 55.958]
  MoveL 159 to (93.53, 73.39, 93.13) mm, rotated rx -127.55 ry 0 rz 129.12 deg; joints [10.174, -48.241, 77.794, -0.913, 57.112, -25.386, 55.683]
  MoveL 160 to (88.83, 73.91, 97.23) mm, rotated rx -129.57 ry 0 rz 130.81 deg; joints [10.582, -48.48, 78.372, -0.857, 57.112, -27.019, 53.658]
  MoveL 161 to (88.79, 73.91, 97.27) mm, rotated rx -129.72 ry 0 rz 130.91 deg; joints [10.603, -48.482, 78.402, -0.851, 57.112, -27.157, 53.526]
  MoveL 162 to (87.4, 73.49, 98.82) mm, rotated rx -130.61 ry 0 rz 131.26 deg; joints [10.771, -48.583, 78.654, -0.823, 57.112, -27.886, 53.025]
  MoveL 163 to (87.43, 73.5, 98.79) mm, rotated rx -131.37 ry 0 rz 131.12 deg; joints [10.865, -48.659, 78.796, -0.811, 57.112, -28.556, 53.097]
  MoveL 164 to (87.12, 70.77, 101.04) mm, rotated rx -132.5 ry 0 rz 130.18 deg; joints [11.09, -48.808, 79.146, -0.771, 57.112, -29.482, 53.837]
  MoveL 165 to (86.99, 70.33, 101.46) mm, rotated rx -132.5 ry 0 rz 130.18 deg; joints [11.105, -48.805, 79.17, -0.765, 57.112, -29.47, 53.809]
  MoveL 166 to (86.3, 69.7, 102.47) mm, rotated rx -132.5 ry 0 rz 130.18 deg; joints [11.144, -48.83, 79.232, -0.757, 57.112, -29.435, 53.771]
  MoveL 167 to (86.12, 69.64, 102.67) mm, rotated rx -132.6 ry 0 rz 130.21 deg; joints [11.164, -48.844, 79.264, -0.753, 57.112, -29.52, 53.716]
  MoveL 168 to (85.06, 69.65, 103.54) mm, rotated rx -132.6 ry 0 rz 130.21 deg; joints [11.199, -48.898, 79.313, -0.753, 57.126, -29.485, 53.71]
  MoveL 169 to (83.74, 70.04, 104.35) mm, rotated rx -133.03 ry 0 rz 130.82 deg; joints [11.283, -48.957, 79.449, -0.737, 57.126, -29.838, 53.023]
  MoveL 170 to (83.76, 70.05, 104.32) mm, rotated rx -133.57 ry 0 rz 131.2 deg; joints [11.346, -48.963, 79.554, -0.713, 57.126, -30.328, 52.536]
  MoveL 171 to (82.94, 69.61, 105.27) mm, rotated rx -134.23 ry 0 rz 131.33 deg; joints [11.463, -49.047, 79.748, -0.688, 57.126, -30.883, 52.304]
  MoveL 172 to (82.78, 69.45, 105.51) mm, rotated rx -134.36 ry 0 rz 131.32 deg; joints [11.487, -49.065, 79.789, -0.683, 57.126, -30.987, 52.286]
  MoveL 173 to (81.07, 67.48, 108.08) mm, rotated rx -135.8 ry 0 rz 131.12 deg; joints [11.761, -49.275, 80.26, -0.623, 57.126, -32.186, 52.217]
  MoveL 174 to (91.57, 76.65, 122.42) mm, rotated rx -135.8 ry 0 rz 131.12 deg; joints [12.165, -48.59, 78.742, -0.882, 57.126, -31.652, 53.08]
  Set speed (1000.0 mm/s)
  MoveL 175 to (90.79, 72.41, 125.54) mm, rotated rx -137.12 ry 0 rz 129.8 deg; joints [12.444, -48.808, 79.243, -0.815, 57.126, -32.724, 54.119]
  Set speed (5.0 mm/s)
  MoveL 176 to (80.33, 63.7, 110.89) mm, rotated rx -137.12 ry 0 rz 129.8 deg; joints [12.029, -49.492, 80.739, -0.559, 57.126, -33.269, 53.277]
  Set speed (16.7 mm/s)
  MoveL 177 to (78.53, 62.71, 112.72) mm, rotated rx -138.15 ry 0 rz 130.02 deg; joints [12.224, -49.657, 81.101, -0.509, 57.126, -34.137, 52.852]
  MoveL 178 to (77.97, 61.99, 113.51) mm, rotated rx -138.89 ry 0 rz 129.9 deg; joints [12.342, -49.76, 81.323, -0.477, 57.126, -34.769, 52.845]
  MoveL 179 to (77.39, 61.55, 114.14) mm, rotated rx -138.89 ry 0 rz 129.9 deg; joints [12.368, -49.785, 81.372, -0.471, 57.126, -34.746, 52.82]
  MoveL 180 to (77.25, 61.49, 114.27) mm, rotated rx -138.96 ry 0 rz 129.93 deg; joints [12.382, -49.798, 81.399, -0.467, 57.126, -34.81, 52.778]
  MoveL 181 to (76.96, 61.41, 114.51) mm, rotated rx -138.96 ry 0 rz 129.93 deg; joints [12.392, -49.812, 81.418, -0.466, 57.126, -34.8, 52.774]
  MoveL 182 to (76.39, 61.28, 114.96) mm, rotated rx -139.22 ry 0 rz 130.09 deg; joints [12.44, -49.856, 81.512, -0.453, 57.126, -35.022, 52.56]
  MoveL 183 to (76.36, 61.31, 114.96) mm, rotated rx -140.09 ry 0 rz 130 deg; joints [12.54, -49.958, 81.706, -0.428, 57.126, -35.796, 52.564]
  MoveL 184 to (75.89, 58.95, 116.5) mm, rotated rx -140.99 ry 0 rz 129.11 deg; joints [12.706, -50.113, 82.037, -0.379, 57.126, -36.557, 53.27]
  MoveL 185 to (75.88, 58.99, 116.48) mm, rotated rx -141.42 ry 0 rz 128.03 deg; joints [12.757, -50.233, 82.107, -0.379, 57.178, -36.935, 54.349]
  MoveL 186 to (78.23, 55.19, 116.8) mm, rotated rx -141.6 ry 0 rz 125.37 deg; joints [12.791, -50.266, 82.176, -0.369, 57.178, -37.092, 56.972]
  MoveL 187 to (78.45, 54.73, 116.87) mm, rotated rx -141.6 ry 0 rz 125.37 deg; joints [12.792, -50.241, 82.182, -0.36, 57.178, -37.096, 56.941]
  MoveL 188 to (78.6, 54.34, 116.95) mm, rotated rx -141.65 ry 0 rz 125.13 deg; joints [12.801, -50.25, 82.2, -0.357, 57.178, -37.137, 57.173]
  MoveL 189 to (78.73, 53.86, 117.08) mm, rotated rx -141.65 ry 0 rz 125.13 deg; joints [12.805, -50.23, 82.211, -0.347, 57.179, -37.138, 57.14]
  MoveL 190 to (79.04, 52.14, 117.64) mm, rotated rx -141.99 ry 0 rz 124.18 deg; joints [12.867, -50.29, 82.338, -0.328, 57.179, -37.428, 58.021]
  MoveL 191 to (79, 52.2, 117.64) mm, rotated rx -141.9 ry 0 rz 122.48 deg; joints [12.865, -50.435, 82.318, -0.379, 57.178, -37.307, 59.893]
  MoveL 192 to (80.03, 51.74, 117.15) mm, rotated rx -141.6 ry 0 rz 121.92 deg; joints [12.811, -50.383, 82.208, -0.395, 57.178, -37.058, 60.512]
  MoveL 193 to (80.55, 51.42, 116.94) mm, rotated rx -141.6 ry 0 rz 121.92 deg; joints [12.802, -50.354, 82.199, -0.395, 57.158, -37.068, 60.512]
  MoveL 194 to (80.84, 51.2, 116.84) mm, rotated rx -141.54 ry 0 rz 121.71 deg; joints [12.791, -50.343, 82.177, -0.398, 57.158, -37.018, 60.727]
  MoveL 195 to (81.31, 50.73, 116.71) mm, rotated rx -141.54 ry 0 rz 121.71 deg; joints [12.785, -50.314, 82.177, -0.396, 57.136, -37.025, 60.719]
  MoveL 196 to (83.31, 48.21, 116.37) mm, rotated rx -141.34 ry 0 rz 119.81 deg; joints [12.748, -50.279, 82.103, -0.407, 57.136, -36.855, 62.663]
  MoveL 197 to (83.12, 48.42, 116.42) mm, rotated rx -141.33 ry 0 rz 119.71 deg; joints [12.75, -50.301, 82.103, -0.413, 57.139, -36.836, 62.779]
  MoveL 198 to (83.31, 48.23, 116.36) mm, rotated rx -141.29 ry 0 rz 119.56 deg; joints [12.744, -50.296, 82.091, -0.415, 57.139, -36.808, 62.936]
  MoveL 199 to (85.09, 46.58, 115.75) mm, rotated rx -140.91 ry 0 rz 118.12 deg; joints [12.675, -50.237, 81.952, -0.437, 57.139, -36.48, 64.46]
  MoveL 200 to (85.39, 46.24, 115.66) mm, rotated rx -140.91 ry 0 rz 118.12 deg; joints [12.671, -50.217, 81.952, -0.436, 57.123, -36.485, 64.455]
  MoveL 201 to (85.89, 45.32, 115.66) mm, rotated rx -140.91 ry 0 rz 118.12 deg; joints [12.668, -50.161, 81.952, -0.42, 57.121, -36.496, 64.4]
  MoveL 202 to (85.97, 45.07, 115.69) mm, rotated rx -140.93 ry 0 rz 117.97 deg; joints [12.671, -50.164, 81.96, -0.419, 57.121, -36.513, 64.548]
  MoveL 203 to (86.13, 44.14, 115.93) mm, rotated rx -140.93 ry 0 rz 117.97 deg; joints [12.679, -50.125, 81.979, -0.401, 57.121, -36.515, 64.487]
  MoveL 204 to (86.12, 43.12, 116.32) mm, rotated rx -141.16 ry 0 rz 117.44 deg; joints [12.721, -50.165, 82.064, -0.388, 57.121, -36.709, 64.974]
  MoveL 205 to (86.12, 43.1, 116.33) mm, rotated rx -141.3 ry 0 rz 116.24 deg; joints [12.74, -50.256, 82.064, -0.396, 57.188, -36.829, 66.197]
  MoveL 206 to (86.62, 42.44, 116.21) mm, rotated rx -141.23 ry 0 rz 115.75 deg; joints [12.726, -50.243, 82.037, -0.4, 57.188, -36.767, 66.696]
  MoveL 207 to (86.79, 42.19, 116.17) mm, rotated rx -141.23 ry 0 rz 115.75 deg; joints [12.724, -50.23, 82.038, -0.398, 57.18, -36.77, 66.689]
  MoveL 208 to (87.08, 41.69, 116.13) mm, rotated rx -141.2 ry 0 rz 115.42 deg; joints [12.72, -50.226, 82.029, -0.399, 57.18, -36.75, 67.032]
  MoveL 209 to (87.25, 41.36, 116.12) mm, rotated rx -141.2 ry 0 rz 115.42 deg; joints [12.719, -50.206, 82.029, -0.394, 57.178, -36.754, 67.014]
  MoveL 210 to (89.56, 35.65, 116.25) mm, rotated rx -141.28 ry 0 rz 111.76 deg; joints [12.733, -50.22, 82.057, -0.39, 57.178, -36.819, 70.658]
  MoveL 211 to (89.72, 35.04, 116.32) mm, rotated rx -141.28 ry 0 rz 111.76 deg; joints [12.734, -50.188, 82.062, -0.379, 57.178, -36.824, 70.62]
  MoveL 212 to (89.79, 34.57, 116.4) mm, rotated rx -141.33 ry 0 rz 111.48 deg; joints [12.743, -50.197, 82.081, -0.376, 57.178, -36.868, 70.891]
  MoveL 213 to (89.82, 34.13, 116.51) mm, rotated rx -141.33 ry 0 rz 111.48 deg; joints [12.746, -50.179, 82.09, -0.368, 57.178, -36.87, 70.863]
  MoveL 214 to (89.71, 29.88, 117.75) mm, rotated rx -142.08 ry 0 rz 109.12 deg; joints [12.882, -50.311, 82.368, -0.326, 57.178, -37.502, 73.072]
  MoveL 215 to (89.69, 29.71, 117.82) mm, rotated rx -142.2 ry 0 rz 108.68 deg; joints [12.898, -50.35, 82.393, -0.326, 57.193, -37.602, 73.512]
  MoveL 216 to (90.3, 24.27, 118.59) mm, rotated rx -142.67 ry 0 rz 105.4 deg; joints [12.983, -50.434, 82.57, -0.299, 57.193, -38.003, 76.696]
  MoveL 217 to (90.61, 17.61, 119.53) mm, rotated rx -143.25 ry 0 rz 101.36 deg; joints [13.088, -50.54, 82.79, -0.265, 57.193, -38.497, 80.615]
  MoveL 218 to (90.33, 16.36, 119.92) mm, rotated rx -143.25 ry 0 rz 101.36 deg; joints [13.101, -50.494, 82.825, -0.24, 57.193, -38.497, 80.531]
  MoveL 219 to (89.52, 15.51, 120.64) mm, rotated rx -143.25 ry 0 rz 101.36 deg; joints [13.129, -50.49, 82.891, -0.218, 57.193, -38.48, 80.458]
  MoveL 220 to (88.71, 15.31, 121.26) mm, rotated rx -143.25 ry 0 rz 101.36 deg; joints [13.156, -50.516, 82.948, -0.209, 57.193, -38.458, 80.426]
  MoveL 221 to (87.75, 15.63, 121.92) mm, rotated rx -143.25 ry 0 rz 101.36 deg; joints [13.185, -50.572, 83.008, -0.208, 57.193, -38.429, 80.422]
  MoveL 222 to (87.03, 16.36, 122.33) mm, rotated rx -143.25 ry 0 rz 101.36 deg; joints [13.204, -50.623, 83.032, -0.208, 57.221, -38.411, 80.422]
  MoveL 223 to (86.62, 17.37, 122.48) mm, rotated rx -143.25 ry 0 rz 101.36 deg; joints [13.212, -50.674, 83.032, -0.215, 57.249, -38.398, 80.447]
  MoveL 224 to (85.75, 21.09, 122.51) mm, rotated rx -143.27 ry 0 rz 103.84 deg; joints [13.215, -50.678, 83.039, -0.214, 57.249, -38.414, 77.967]
  MoveL 225 to (84.62, 25.11, 122.54) mm, rotated rx -143.29 ry 0 rz 106.55 deg; joints [13.219, -50.682, 83.047, -0.213, 57.249, -38.431, 75.254]
  MoveL 226 to (84.64, 25.05, 122.54) mm, rotated rx -143.41 ry 0 rz 107.29 deg; joints [13.229, -50.631, 83.077, -0.188, 57.249, -38.56, 74.424]
  MoveL 227 to (82.86, 26.95, 123.35) mm, rotated rx -143.94 ry 0 rz 108.84 deg; joints [13.323, -50.732, 83.283, -0.155, 57.249, -39.015, 72.763]
  MoveL 228 to (82.69, 27.15, 123.42) mm, rotated rx -143.94 ry 0 rz 108.84 deg; joints [13.326, -50.743, 83.284, -0.155, 57.258, -39.012, 72.763]
  MoveL 229 to (82.43, 27.47, 123.52) mm, rotated rx -144.01 ry 0 rz 109.1 deg; joints [13.338, -50.756, 83.31, -0.151, 57.258, -39.069, 72.493]
  MoveL 230 to (80.51, 29.65, 124.28) mm, rotated rx -144.53 ry 0 rz 110.94 deg; joints [13.428, -50.851, 83.512, -0.118, 57.258, -39.517, 70.54]
  MoveL 231 to (91.35, 33.8, 140.57) mm, rotated rx -144.53 ry 0 rz 110.94 deg; joints [13.903, -50.184, 82.153, -0.346, 57.258, -38.921, 71.258]
  Set speed (1000.0 mm/s)
  MoveL 232 to (87.3, 33, 143.31) mm, rotated rx -146.24 ry 0 rz 111.57 deg; joints [14.207, -50.506, 82.853, -0.225, 57.258, -40.388, 70.237]
  Set speed (5.0 mm/s)
  MoveL 233 to (76.96, 28.91, 126.68) mm, rotated rx -146.24 ry 0 rz 111.57 deg; joints [13.718, -51.167, 84.179, -0.005, 57.258, -40.995, 69.547]
  Set speed (16.7 mm/s)
  MoveL 234 to (74.45, 30.84, 127.73) mm, rotated rx -146.98 ry 0 rz 113.52 deg; joints [13.844, -51.317, 84.477, 0.044, 57.258, -41.636, 67.45]
  MoveL 235 to (73.91, 31.36, 127.91) mm, rotated rx -146.98 ry 0 rz 113.52 deg; joints [13.853, -51.351, 84.481, 0.044, 57.288, -41.628, 67.45]
  MoveL 236 to (73.69, 31.64, 127.97) mm, rotated rx -147.02 ry 0 rz 113.76 deg; joints [13.86, -51.359, 84.498, 0.047, 57.288, -41.663, 67.197]
  MoveL 237 to (73.56, 31.82, 128) mm, rotated rx -147.02 ry 0 rz 113.76 deg; joints [13.862, -51.369, 84.498, 0.046, 57.293, -41.661, 67.202]
  MoveL 238 to (71.61, 34.59, 128.39) mm, rotated rx -147.3 ry 0 rz 116.16 deg; joints [13.909, -51.427, 84.611, 0.064, 57.293, -41.902, 64.748]
  MoveL 239 to (71.26, 35.29, 128.38) mm, rotated rx -148.41 ry 0 rz 118.12 deg; joints [14.02, -51.472, 84.9, 0.146, 57.293, -42.947, 62.531]
  MoveL 240 to (70.59, 34.73, 128.91) mm, rotated rx -148.79 ry 0 rz 117.99 deg; joints [14.084, -51.552, 85.056, 0.172, 57.293, -43.277, 62.587]
  MoveL 241 to (70.2, 34.48, 129.19) mm, rotated rx -148.79 ry 0 rz 117.99 deg; joints [14.097, -51.567, 85.088, 0.178, 57.293, -43.268, 62.569]
  MoveL 242 to (69.17, 34.3, 129.79) mm, rotated rx -148.79 ry 0 rz 117.99 deg; joints [14.125, -51.62, 85.156, 0.184, 57.294, -43.242, 62.553]
  MoveL 243 to (68.72, 34.35, 130.02) mm, rotated rx -148.96 ry 0 rz 118.17 deg; joints [14.153, -51.655, 85.225, 0.196, 57.294, -43.388, 62.331]
  MoveL 244 to (68.28, 34.44, 130.23) mm, rotated rx -148.96 ry 0 rz 118.17 deg; joints [14.163, -51.682, 85.247, 0.196, 57.298, -43.378, 62.331]
  MoveL 245 to (67.34, 35, 130.57) mm, rotated rx -148.96 ry 0 rz 118.17 deg; joints [14.18, -51.736, 85.268, 0.196, 57.331, -43.361, 62.331]
  MoveL 246 to (64.99, 37.06, 131.19) mm, rotated rx -149.43 ry 0 rz 120.42 deg; joints [14.258, -51.837, 85.464, 0.229, 57.331, -43.773, 59.981]
  MoveL 247 to (64.7, 37.38, 131.24) mm, rotated rx -149.48 ry 0 rz 120.77 deg; joints [14.265, -51.846, 85.484, 0.233, 57.331, -43.816, 59.627]
  MoveL 248 to (62.31, 39.22, 131.86) mm, rotated rx -149.95 ry 0 rz 122.96 deg; joints [14.343, -51.95, 85.683, 0.267, 57.331, -44.233, 57.334]
  MoveL 249 to (61.89, 39.47, 131.98) mm, rotated rx -150.04 ry 0 rz 123.24 deg; joints [14.358, -51.974, 85.72, 0.272, 57.331, -44.305, 57.046]
  MoveL 250 to (59.39, 41.33, 132.56) mm, rotated rx -150.49 ry 0 rz 125.57 deg; joints [14.432, -52.075, 85.913, 0.304, 57.331, -44.705, 54.618]
  MoveL 251 to (59.02, 41.65, 132.62) mm, rotated rx -150.53 ry 0 rz 125.84 deg; joints [14.439, -52.09, 85.929, 0.305, 57.332, -44.732, 54.342]
  MoveL 252 to (56.54, 43.48, 133.11) mm, rotated rx -150.92 ry 0 rz 128.21 deg; joints [14.502, -52.178, 86.095, 0.333, 57.332, -45.077, 51.894]
  MoveL 253 to (56.15, 43.82, 133.17) mm, rotated rx -150.92 ry 0 rz 128.21 deg; joints [14.506, -52.203, 86.095, 0.329, 57.343, -45.071, 51.907]
  MoveL 254 to (55.97, 44, 133.19) mm, rotated rx -150.93 ry 0 rz 128.41 deg; joints [14.508, -52.205, 86.101, 0.33, 57.343, -45.082, 51.702]
  MoveL 255 to (54.6, 45.38, 133.29) mm, rotated rx -151.01 ry 0 rz 129.95 deg; joints [14.521, -52.226, 86.136, 0.336, 57.343, -45.154, 50.145]
  MoveL 256 to (52.84, 46.44, 133.63) mm, rotated rx -151.34 ry 0 rz 132 deg; joints [14.569, -52.267, 86.27, 0.369, 57.343, -45.455, 48.004]
  MoveL 257 to (51.9, 47.35, 133.68) mm, rotated rx -151.34 ry 0 rz 132 deg; joints [14.575, -52.335, 86.27, 0.348, 57.35, -45.437, 48.068]
  MoveL 258 to (51.82, 47.48, 133.67) mm, rotated rx -151.33 ry 0 rz 132.12 deg; joints [14.574, -52.333, 86.265, 0.347, 57.35, -45.428, 47.944]
  MoveL 259 to (51.47, 48.26, 133.53) mm, rotated rx -151.33 ry 0 rz 132.12 deg; joints [14.569, -52.365, 86.245, 0.329, 57.35, -45.422, 47.999]
  MoveL 260 to (51.2, 49.25, 133.27) mm, rotated rx -151.12 ry 0 rz 132.87 deg; joints [14.535, -52.317, 86.156, 0.314, 57.35, -45.238, 47.293]
  MoveL 261 to (51.21, 49.21, 133.27) mm, rotated rx -151 ry 0 rz 133.71 deg; joints [14.522, -52.264, 86.148, 0.314, 57.305, -45.127, 46.452]
  MoveL 262 to (50.57, 49.97, 133.24) mm, rotated rx -150.97 ry 0 rz 134.5 deg; joints [14.518, -52.257, 86.136, 0.312, 57.305, -45.102, 45.666]
  MoveL 263 to (50.14, 50.63, 133.15) mm, rotated rx -150.97 ry 0 rz 134.5 deg; joints [14.516, -52.292, 86.123, 0.295, 57.305, -45.095, 45.715]
  MoveL 264 to (49.96, 51.08, 133.05) mm, rotated rx -150.95 ry 0 rz 134.6 deg; joints [14.51, -52.299, 86.104, 0.286, 57.305, -45.077, 45.645]
  MoveL 265 to (49.78, 51.65, 132.89) mm, rotated rx -150.83 ry 0 rz 135.03 deg; joints [14.49, -52.271, 86.052, 0.278, 57.305, -44.968, 45.246]
  MoveL 266 to (49.8, 51.61, 132.9) mm, rotated rx -150.7 ry 0 rz 136.06 deg; joints [14.476, -52.209, 86.048, 0.278, 57.247, -44.85, 44.214]
  MoveL 267 to (48.92, 52.42, 132.91) mm, rotated rx -150.71 ry 0 rz 137.01 deg; joints [14.478, -52.211, 86.052, 0.278, 57.247, -44.858, 43.258]
  MoveL 268 to (48.42, 53.02, 132.86) mm, rotated rx -150.71 ry 0 rz 137.01 deg; joints [14.477, -52.248, 86.044, 0.263, 57.247, -44.85, 43.306]
  MoveL 269 to (48.33, 53.17, 132.83) mm, rotated rx -150.69 ry 0 rz 137.15 deg; joints [14.474, -52.244, 86.035, 0.261, 57.247, -44.832, 43.175]
  MoveL 270 to (48.11, 53.58, 132.75) mm, rotated rx -150.69 ry 0 rz 137.15 deg; joints [14.471, -52.261, 86.023, 0.251, 57.247, -44.829, 43.206]
  MoveL 271 to (47.66, 54.65, 132.47) mm, rotated rx -150.47 ry 0 rz 137.98 deg; joints [14.436, -52.212, 85.932, 0.236, 57.247, -44.639, 42.414]
  MoveL 272 to (47.68, 54.65, 132.47) mm, rotated rx -150.36 ry 0 rz 138.58 deg; joints [14.425, -52.17, 85.919, 0.236, 57.218, -44.547, 41.811]
  MoveL 273 to (45.09, 57.02, 132.37) mm, rotated rx -150.28 ry 0 rz 141.55 deg; joints [14.411, -52.139, 85.886, 0.235, 57.218, -44.475, 38.851]
  MoveL 274 to (44.64, 57.53, 132.31) mm, rotated rx -150.28 ry 0 rz 141.55 deg; joints [14.41, -52.17, 85.876, 0.221, 57.218, -44.469, 38.893]
  MoveL 275 to (44.55, 57.65, 132.28) mm, rotated rx -150.26 ry 0 rz 141.66 deg; joints [14.406, -52.165, 85.868, 0.22, 57.218, -44.451, 38.782]
  MoveL 276 to (44.4, 57.89, 132.23) mm, rotated rx -150.26 ry 0 rz 141.66 deg; joints [14.405, -52.176, 85.861, 0.214, 57.218, -44.45, 38.8]
  MoveL 277 to (43.89, 58.79, 132) mm, rotated rx -150.08 ry 0 rz 142.42 deg; joints [14.375, -52.136, 85.785, 0.201, 57.218, -44.293, 38.082]
  MoveL 278 to (43.93, 58.75, 132) mm, rotated rx -149.99 ry 0 rz 143.07 deg; joints [14.366, -52.094, 85.783, 0.201, 57.179, -44.213, 37.43]
  MoveL 279 to (43.1, 59.45, 131.97) mm, rotated rx -149.96 ry 0 rz 143.92 deg; joints [14.361, -52.087, 85.77, 0.199, 57.179, -44.186, 36.587]
  MoveL 280 to (42.55, 60.06, 131.87) mm, rotated rx -149.96 ry 0 rz 143.92 deg; joints [14.359, -52.124, 85.757, 0.182, 57.179, -44.179, 36.638]
  MoveL 281 to (42.43, 60.25, 131.82) mm, rotated rx -149.93 ry 0 rz 144.08 deg; joints [14.353, -52.116, 85.743, 0.18, 57.179, -44.149, 36.486]
  MoveL 282 to (42.18, 60.7, 131.69) mm, rotated rx -149.93 ry 0 rz 144.08 deg; joints [14.348, -52.132, 85.726, 0.169, 57.179, -44.148, 36.52]
  MoveL 283 to (41.74, 61.75, 131.34) mm, rotated rx -149.66 ry 0 rz 144.84 deg; joints [14.304, -52.073, 85.614, 0.15, 57.179, -43.912, 35.816]
  MoveL 284 to (41.74, 61.75, 131.34) mm, rotated rx -149.52 ry 0 rz 146.47 deg; joints [14.287, -51.973, 85.614, 0.161, 57.11, -43.795, 34.149]
  MoveL 285 to (38.81, 62.72, 131.78) mm, rotated rx -149.85 ry 0 rz 148.79 deg; joints [14.343, -52.046, 85.755, 0.185, 57.11, -44.091, 31.755]
  MoveL 286 to (38.37, 62.9, 131.83) mm, rotated rx -149.85 ry 0 rz 148.79 deg; joints [14.346, -52.069, 85.755, 0.18, 57.12, -44.086, 31.77]
  MoveL 287 to (38.1, 63.04, 131.84) mm, rotated rx -149.87 ry 0 rz 149.03 deg; joints [14.347, -52.072, 85.76, 0.181, 57.12, -44.095, 31.529]
  MoveL 288 to (35.74, 64.17, 131.95) mm, rotated rx -149.95 ry 0 rz 151.05 deg; joints [14.362, -52.092, 85.797, 0.187, 57.12, -44.171, 29.495]
  MoveL 289 to (33.28, 64.63, 132.38) mm, rotated rx -150.33 ry 0 rz 153.4 deg; joints [14.419, -52.14, 85.95, 0.223, 57.12, -44.514, 27.036]
  MoveL 290 to (32.52, 64.87, 132.44) mm, rotated rx -150.33 ry 0 rz 153.4 deg; joints [14.424, -52.18, 85.95, 0.215, 57.133, -44.505, 27.063]
  MoveL 291 to (31.84, 65.29, 132.4) mm, rotated rx -150.44 ry 0 rz 154.99 deg; joints [14.429, -52.128, 85.976, 0.241, 57.133, -44.617, 25.387]
  MoveL 292 to (31.04, 65.26, 132.61) mm, rotated rx -150.6 ry 0 rz 155.56 deg; joints [14.455, -52.164, 86.045, 0.253, 57.133, -44.761, 24.785]
  MoveL 293 to (35.1, 74.19, 150.04) mm, rotated rx -150.6 ry 0 rz 155.56 deg; joints [14.979, -51.524, 84.811, 0.055, 57.133, -44.129, 25.402]
  Set speed (1000.0 mm/s)
  MoveL 294 to (31.87, 77.18, 149.24) mm, rotated rx -149.94 ry 0 rz 157.44 deg; joints [14.878, -51.46, 84.537, -0.019, 57.133, -43.528, 23.741]
  Set speed (5.0 mm/s)
  MoveL 295 to (28.02, 67.93, 131.93) mm, rotated rx -149.94 ry 0 rz 157.44 deg; joints [14.36, -52.103, 85.784, 0.183, 57.133, -44.157, 23.114]
  Set speed (16.7 mm/s)
  MoveL 296 to (27.16, 68.34, 131.9) mm, rotated rx -149.91 ry 0 rz 158.19 deg; joints [14.356, -52.097, 85.772, 0.181, 57.133, -44.133, 22.369]
  MoveL 297 to (26.15, 68.55, 132) mm, rotated rx -150 ry 0 rz 159.46 deg; joints [14.367, -52.084, 85.808, 0.198, 57.133, -44.218, 21.052]
  MoveL 298 to (29.66, 77.92, 149.32) mm, rotated rx -150 ry 0 rz 159.46 deg; joints [14.886, -51.441, 84.562, -0.004, 57.133, -43.589, 21.678]
  Set speed (1000.0 mm/s)
  MoveL 299 to (28.49, 75.29, 150.89) mm, rotated rx -151.46 ry 0 rz 160.75 deg; joints [15.104, -51.656, 85.15, 0.13, 57.133, -44.905, 20.003]
  Set speed (5.0 mm/s)
  MoveL 300 to (25.34, 66.27, 133.32) mm, rotated rx -151.46 ry 0 rz 160.75 deg; joints [14.574, -52.291, 86.366, 0.322, 57.133, -45.541, 19.399]
  Set speed (16.7 mm/s)
  MoveL 301 to (22.18, 64.04, 134.96) mm, rotated rx -152.84 ry 0 rz 162.67 deg; joints [14.791, -52.605, 86.955, 0.424, 57.133, -46.756, 17.185]
  MoveL 302 to (21.45, 63.67, 135.25) mm, rotated rx -152.84 ry 0 rz 162.67 deg; joints [14.806, -52.651, 86.986, 0.424, 57.147, -46.74, 17.185]
  MoveL 303 to (21.08, 63.56, 135.36) mm, rotated rx -152.93 ry 0 rz 162.95 deg; joints [14.821, -52.673, 87.028, 0.431, 57.147, -46.826, 16.889]
  MoveL 304 to (17.76, 62.26, 136.44) mm, rotated rx -153.9 ry 0 rz 165.52 deg; joints [14.97, -52.895, 87.445, 0.505, 57.147, -47.688, 14.114]
  MoveL 305 to (16.46, 62.07, 136.69) mm, rotated rx -153.9 ry 0 rz 165.52 deg; joints [14.983, -52.954, 87.452, 0.505, 57.199, -47.674, 14.115]
  MoveL 306 to (16.13, 62.1, 136.71) mm, rotated rx -153.92 ry 0 rz 165.81 deg; joints [14.986, -52.959, 87.461, 0.506, 57.199, -47.693, 13.824]
  MoveL 307 to (15.19, 62.37, 136.7) mm, rotated rx -153.92 ry 0 rz 165.81 deg; joints [14.989, -53.009, 87.456, 0.487, 57.199, -47.68, 13.88]
  MoveL 308 to (12.24, 63.71, 136.37) mm, rotated rx -153.63 ry 0 rz 168.63 deg; joints [14.944, -52.94, 87.331, 0.466, 57.199, -47.425, 11.113]
  MoveL 309 to (10.77, 64.05, 136.34) mm, rotated rx -153.58 ry 0 rz 170.33 deg; joints [14.937, -52.914, 87.319, 0.466, 57.185, -47.379, 9.418]
  MoveL 310 to (9.59, 64.64, 136.15) mm, rotated rx -153.58 ry 0 rz 170.33 deg; joints [14.931, -52.964, 87.289, 0.437, 57.185, -47.369, 9.502]
  MoveL 311 to (9.4, 64.8, 136.09) mm, rotated rx -153.52 ry 0 rz 170.52 deg; joints [14.922, -52.95, 87.264, 0.433, 57.185, -47.318, 9.323]
  MoveL 312 to (8.95, 65.31, 135.87) mm, rotated rx -153.52 ry 0 rz 170.52 deg; joints [14.913, -52.961, 87.233, 0.418, 57.185, -47.319, 9.367]
  MoveL 313 to (8.07, 66.63, 135.28) mm, rotated rx -153.01 ry 0 rz 171.46 deg; joints [14.834, -52.841, 87.012, 0.381, 57.185, -46.868, 8.534]
  MoveL 314 to (8.08, 66.6, 135.3) mm, rotated rx -152.7 ry 0 rz 172.59 deg; joints [14.801, -52.74, 86.948, 0.38, 57.151, -46.587, 7.393]
  MoveL 315 to (7.87, 66.7, 135.26) mm, rotated rx -152.65 ry 0 rz 173.37 deg; joints [14.794, -52.707, 86.945, 0.381, 57.121, -46.541, 6.612]
  MoveL 316 to (6.44, 66.79, 135.3) mm, rotated rx -152.68 ry 0 rz 174.59 deg; joints [14.798, -52.714, 86.957, 0.382, 57.121, -46.566, 5.393]
  MoveL 317 to (4.06, 66.43, 135.57) mm, rotated rx -152.94 ry 0 rz 177.1 deg; joints [14.836, -52.744, 87.068, 0.412, 57.121, -46.811, 2.797]
  MoveL 318 to (3.18, 66.36, 135.62) mm, rotated rx -152.95 ry 0 rz 177.19 deg; joints [14.842, -52.786, 87.074, 0.402, 57.128, -46.811, 2.741]
  MoveL 319 to (2.64, 66.4, 135.61) mm, rotated rx -152.95 ry 0 rz 177.65 deg; joints [14.841, -52.785, 87.071, 0.401, 57.128, -46.805, 2.275]
  MoveL 320 to (2.34, 66.35, 135.64) mm, rotated rx -152.98 ry 0 rz 178.22 deg; joints [14.844, -52.773, 87.084, 0.41, 57.128, -46.836, 1.687]
  MoveL 321 to (0.65, 66.22, 135.73) mm, rotated rx -153.05 ry 0 rz 179.68 deg; joints [14.856, -52.79, 87.115, 0.415, 57.128, -46.9, 0.211]
  MoveL 322 to (0.7, 75.28, 153.55) mm, rotated rx -153.05 ry 0 rz 179.68 deg; joints [15.399, -52.164, 85.935, 0.232, 57.128, -46.256, 0.787]
  Set speed (1000.0 mm/s)
  MoveL 323 to (0.38, 81.25, 150.48) mm, rotated rx -151.91 ry 0 rz 178.05 deg; joints [15.144, -51.927, 85.214, 0.055, 57.128, -45.273, 2.921]
  Set speed (5.0 mm/s)
  MoveL 324 to (0.06, 71.84, 132.84) mm, rotated rx -151.91 ry 0 rz 178.05 deg; joints [14.609, -52.556, 86.416, 0.248, 57.128, -45.913, 2.325]
  Set speed (16.7 mm/s)
  MoveL 325 to (0.46, 72.78, 132.32) mm, rotated rx -151.5 ry 0 rz 177.76 deg; joints [14.544, -52.464, 86.244, 0.218, 57.128, -45.557, 2.693]
  MoveL 326 to (0.48, 72.81, 132.3) mm, rotated rx -150.69 ry 0 rz 177.94 deg; joints [14.46, -52.337, 86.027, 0.186, 57.128, -44.809, 2.61]
  MoveL 327 to (-0.2, 73.83, 131.74) mm, rotated rx -150.24 ry 0 rz 178.5 deg; joints [14.388, -52.238, 85.839, 0.155, 57.128, -44.417, 2.142]
  MoveL 328 to (-0.16, 73.8, 131.76) mm, rotated rx -149.91 ry 0 rz -178.98 deg; joints [14.352, -52.084, 85.828, 0.155, 56.986, -44.118, -0.38]
  MoveL 329 to (-0.94, 73.43, 131.96) mm, rotated rx -150.07 ry 0 rz -178.37 deg; joints [14.378, -52.118, 85.895, 0.166, 56.986, -44.258, -1.026]
  MoveL 330 to (-1, 73.35, 132.01) mm, rotated rx -151.44 ry 0 rz -177.55 deg; joints [14.516, -52.261, 86.265, 0.247, 56.986, -45.537, -2.083]
  MoveL 331 to (0.11, 71.82, 132.84) mm, rotated rx -152.1 ry 0 rz -178.38 deg; joints [14.622, -52.41, 86.546, 0.295, 56.986, -46.114, -1.389]
  MoveL 332 to (-0.15, 81.18, 150.52) mm, rotated rx -152.1 ry 0 rz -178.38 deg; joints [15.158, -51.781, 85.344, 0.103, 56.986, -45.473, -0.793]
  Set speed (1000.0 mm/s)
  MoveL 333 to (-2.2, 76.44, 152.97) mm, rotated rx -152.72 ry 0 rz -177.39 deg; joints [15.342, -52.084, 85.836, 0.174, 56.986, -45.953, -1.982]
  Set speed (5.0 mm/s)
  MoveL 334 to (-1.78, 67.29, 135.19) mm, rotated rx -152.72 ry 0 rz -177.39 deg; joints [14.802, -52.711, 87.023, 0.36, 56.986, -46.597, -2.564]
  Set speed (16.7 mm/s)
  MoveL 335 to (-4.6, 65.51, 136) mm, rotated rx -153.42 ry 0 rz -174.84 deg; joints [14.911, -52.874, 87.327, 0.413, 56.986, -47.217, -5.254]
  MoveL 336 to (-5.37, 65.15, 136.14) mm, rotated rx -153.42 ry 0 rz -174.84 deg; joints [14.918, -52.91, 87.327, 0.413, 57.022, -47.209, -5.254]
  MoveL 337 to (-5.53, 65.11, 136.15) mm, rotated rx -153.43 ry 0 rz -174.7 deg; joints [14.92, -52.913, 87.332, 0.414, 57.022, -47.221, -5.398]
  MoveL 338 to (-6.84, 65.06, 136.12) mm, rotated rx -153.43 ry 0 rz -174.7 deg; joints [14.923, -52.978, 87.324, 0.388, 57.022, -47.204, -5.321]
  MoveL 339 to (-8.18, 65.31, 135.92) mm, rotated rx -153.26 ry 0 rz -173.56 deg; joints [14.896, -52.937, 87.249, 0.375, 57.022, -47.051, -6.43]
  MoveL 340 to (-8.39, 65.37, 135.88) mm, rotated rx -153.35 ry 0 rz -171.43 deg; joints [14.896, -52.832, 87.275, 0.421, 57.022, -47.17, -8.699]
  MoveL 341 to (-8.77, 65.04, 136.01) mm, rotated rx -153.47 ry 0 rz -171.05 deg; joints [14.914, -52.86, 87.327, 0.43, 57.022, -47.276, -9.095]
  MoveL 342 to (-9.88, 63.93, 136.46) mm, rotated rx -153.9 ry 0 rz -169.84 deg; joints [14.978, -52.953, 87.508, 0.463, 57.022, -47.657, -10.405]
  MoveL 343 to (-10.85, 63.27, 136.7) mm, rotated rx -153.9 ry 0 rz -169.8 deg; joints [14.991, -53.006, 87.517, 0.463, 57.066, -47.641, -10.437]
  MoveL 344 to (-11.5, 63.12, 136.72) mm, rotated rx -153.9 ry 0 rz -169.79 deg; joints [14.993, -53.04, 87.517, 0.452, 57.066, -47.63, -10.419]
  MoveL 345 to (-12.33, 63.14, 136.63) mm, rotated rx -153.89 ry 0 rz -169.77 deg; joints [14.991, -53.074, 87.502, 0.434, 57.066, -47.621, -10.39]
  MoveL 346 to (-13.46, 63.61, 136.31) mm, rotated rx -153.89 ry 0 rz -169.73 deg; joints [14.978, -53.1, 87.453, 0.408, 57.066, -47.617, -10.345]
  MoveL 347 to (-14.09, 64.07, 136.03) mm, rotated rx -153.48 ry 0 rz -168.85 deg; joints [14.922, -52.992, 87.301, 0.391, 57.066, -47.252, -11.186]
  MoveL 348 to (-14.97, 64.39, 135.78) mm, rotated rx -153.26 ry 0 rz -168.14 deg; joints [14.888, -52.94, 87.207, 0.374, 57.066, -47.058, -11.845]
  MoveL 349 to (-15.61, 64.77, 135.53) mm, rotated rx -153 ry 0 rz -165.4 deg; joints [14.847, -52.787, 87.152, 0.374, 56.97, -46.834, -14.587]
  MoveL 350 to (-16.81, 63.7, 135.89) mm, rotated rx -153.32 ry 0 rz -164.14 deg; joints [14.896, -52.861, 87.291, 0.398, 56.97, -47.117, -15.911]
  MoveL 351 to (-17.27, 63.36, 135.99) mm, rotated rx -153.32 ry 0 rz -164.14 deg; joints [14.902, -52.886, 87.292, 0.398, 56.993, -47.112, -15.911]
  MoveL 352 to (-18.51, 62.98, 136.01) mm, rotated rx -153.32 ry 0 rz -164.14 deg; joints [14.906, -52.954, 87.29, 0.374, 56.993, -47.094, -15.839]
  MoveL 353 to (-19.16, 62.99, 135.91) mm, rotated rx -153.3 ry 0 rz -164.04 deg; joints [14.902, -52.972, 87.272, 0.362, 56.993, -47.08, -15.903]
  MoveL 354 to (-19.83, 63.08, 135.77) mm, rotated rx -153.18 ry 0 rz -163.5 deg; joints [14.883, -52.943, 87.22, 0.353, 56.993, -46.974, -16.421]
  MoveL 355 to (-19.77, 63.08, 135.78) mm, rotated rx -153.09 ry 0 rz -162.58 deg; joints [14.873, -52.891, 87.22, 0.355, 56.947, -46.891, -17.348]
  MoveL 356 to (-22.31, 62.21, 135.79) mm, rotated rx -153.1 ry 0 rz -160.25 deg; joints [14.875, -52.894, 87.224, 0.355, 56.947, -46.899, -19.677]
  MoveL 357 to (-23.19, 61.68, 135.89) mm, rotated rx -153.18 ry 0 rz -159.45 deg; joints [14.888, -52.918, 87.26, 0.36, 56.947, -46.971, -20.49]
  MoveL 358 to (-25.79, 60.7, 135.86) mm, rotated rx -153.16 ry 0 rz -157.03 deg; joints [14.884, -52.911, 87.248, 0.358, 56.947, -46.947, -22.906]
  MoveL 359 to (-26.87, 60.51, 135.74) mm, rotated rx -153.16 ry 0 rz -157.03 deg; joints [14.881, -52.957, 87.229, 0.335, 56.947, -46.937, -22.838]
  MoveL 360 to (-27.89, 60.75, 135.42) mm, rotated rx -153.16 ry 0 rz -157.03 deg; joints [14.868, -52.978, 87.184, 0.312, 56.947, -46.937, -22.769]
  MoveL 361 to (-28.22, 60.91, 135.28) mm, rotated rx -153.03 ry 0 rz -156.82 deg; joints [14.849, -52.949, 87.132, 0.303, 56.947, -46.83, -22.954]
  MoveL 362 to (-28.59, 61.14, 135.1) mm, rotated rx -153.03 ry 0 rz -156.82 deg; joints [14.841, -52.949, 87.107, 0.294, 56.947, -46.833, -22.928]
  MoveL 363 to (-30.65, 62.62, 133.96) mm, rotated rx -152.07 ry 0 rz -155.74 deg; joints [14.689, -52.728, 86.694, 0.224, 56.947, -45.982, -23.808]
  MoveL 364 to (-31.61, 62.45, 133.82) mm, rotated rx -151.56 ry 0 rz -154.12 deg; joints [14.628, -52.591, 86.54, 0.217, 56.947, -45.527, -25.411]
  MoveL 365 to (-32.47, 62.54, 133.57) mm, rotated rx -151.53 ry 0 rz -154.02 deg; joints [14.615, -52.602, 86.5, 0.199, 56.947, -45.506, -25.453]
  MoveL 366 to (-33.8, 62.92, 133.06) mm, rotated rx -151.12 ry 0 rz -153.19 deg; joints [14.549, -52.509, 86.324, 0.169, 56.947, -45.141, -26.197]
  MoveL 367 to (-34, 62.93, 133.01) mm, rotated rx -151.03 ry 0 rz -152.96 deg; joints [14.537, -52.486, 86.293, 0.166, 56.947, -45.061, -26.422]
  MoveL 368 to (-35.34, 63.18, 132.54) mm, rotated rx -150.65 ry 0 rz -152.1 deg; joints [14.476, -52.402, 86.135, 0.14, 56.947, -44.731, -27.209]
  MoveL 369 to (-35.85, 63.33, 132.33) mm, rotated rx -150.65 ry 0 rz -152.1 deg; joints [14.468, -52.409, 86.109, 0.128, 56.947, -44.734, -27.175]
  MoveL 370 to (-36.74, 64.05, 131.74) mm, rotated rx -150.65 ry 0 rz -152.1 deg; joints [14.441, -52.394, 86.036, 0.108, 56.947, -44.749, -27.114]
  MoveL 371 to (-36.84, 64.2, 131.64) mm, rotated rx -150.57 ry 0 rz -152.08 deg; joints [14.428, -52.377, 86.002, 0.102, 56.947, -44.678, -27.114]
  MoveL 372 to (-37.14, 64.9, 131.21) mm, rotated rx -150.57 ry 0 rz -152.08 deg; joints [14.407, -52.345, 85.949, 0.095, 56.947, -44.695, -27.092]
  MoveL 373 to (-37.3, 65.85, 130.69) mm, rotated rx -149.85 ry 0 rz -152.36 deg; joints [14.309, -52.218, 85.698, 0.052, 56.947, -44.044, -26.685]
  MoveL 374 to (-37.74, 66.5, 130.23) mm, rotated rx -149.5 ry 0 rz -152.29 deg; joints [14.253, -52.144, 85.556, 0.028, 56.947, -43.745, -26.68]
  MoveL 375 to (-37.7, 66.48, 130.25) mm, rotated rx -148.81 ry 0 rz -151.47 deg; joints [14.178, -51.992, 85.378, 0.019, 56.947, -43.118, -27.478]
  MoveL 376 to (-39.22, 66.48, 129.81) mm, rotated rx -148.47 ry 0 rz -150.47 deg; joints [14.122, -51.92, 85.239, -0.004, 56.947, -42.824, -28.406]
  MoveL 377 to (-39.52, 66.48, 129.71) mm, rotated rx -148.41 ry 0 rz -150.3 deg; joints [14.111, -51.909, 85.214, -0.009, 56.947, -42.772, -28.56]
  MoveL 378 to (-40.34, 66.62, 129.39) mm, rotated rx -148.41 ry 0 rz -150.3 deg; joints [14.099, -51.924, 85.177, -0.026, 56.947, -42.775, -28.506]
  MoveL 379 to (-43.07, 67.55, 128.02) mm, rotated rx -147.41 ry 0 rz -148.91 deg; joints [13.93, -51.715, 84.769, -0.092, 56.947, -41.903, -29.691]
  MoveL 380 to (-43.88, 68.03, 127.49) mm, rotated rx -147.41 ry 0 rz -148.91 deg; joints [13.907, -51.709, 84.711, -0.109, 56.947, -41.916, -29.637]
  MoveL 381 to (-44.34, 68.82, 126.91) mm, rotated rx -147.41 ry 0 rz -148.91 deg; joints [13.881, -51.677, 84.649, -0.119, 56.947, -41.937, -29.605]
  MoveL 382 to (-44.39, 69.01, 126.79) mm, rotated rx -147.32 ry 0 rz -148.95 deg; joints [13.867, -51.66, 84.615, -0.125, 56.947, -41.864, -29.551]
  MoveL 383 to (-44.37, 70.12, 126.18) mm, rotated rx -147.32 ry 0 rz -148.95 deg; joints [13.838, -51.595, 84.55, -0.125, 56.947, -41.893, -29.551]
  MoveL 384 to (-43.57, 72.61, 125.05) mm, rotated rx -146.55 ry 0 rz -150.26 deg; joints [13.705, -51.439, 84.242, -0.174, 56.947, -41.23, -28.076]
  MoveL 385 to (-43.37, 73.06, 124.86) mm, rotated rx -146.55 ry 0 rz -150.26 deg; joints [13.697, -51.414, 84.228, -0.174, 56.934, -41.239, -28.076]
  MoveL 386 to (-43.28, 73.2, 124.8) mm, rotated rx -146.52 ry 0 rz -150.36 deg; joints [13.69, -51.407, 84.214, -0.176, 56.934, -41.208, -27.973]
  MoveL 387 to (-43.07, 73.5, 124.7) mm, rotated rx -146.52 ry 0 rz -150.36 deg; joints [13.685, -51.389, 84.209, -0.176, 56.922, -41.213, -27.973]
  MoveL 388 to (-41.36, 75.58, 124.03) mm, rotated rx -146.07 ry 0 rz -152.02 deg; joints [13.609, -51.301, 84.034, -0.204, 56.922, -40.832, -26.218]
  MoveL 389 to (-40.95, 77.64, 122.89) mm, rotated rx -145.02 ry 0 rz -153.52 deg; joints [13.449, -51.171, 83.667, -0.279, 56.922, -39.903, -24.474]
  MoveL 390 to (-40.13, 80.53, 121.29) mm, rotated rx -144 ry 0 rz -154.8 deg; joints [13.267, -50.975, 83.268, -0.34, 56.922, -39.026, -22.988]
  MoveL 391 to (-45.13, 91.17, 137.47) mm, rotated rx -144 ry 0 rz -154.8 deg; joints [13.74, -50.314, 81.906, -0.577, 56.922, -38.429, -22.258]
  Set speed (1000.0 mm/s)
  MoveL 392 to (-40.64, 95.64, 135.82) mm, rotated rx -143.37 ry 0 rz -156.54 deg; joints [13.592, -50.022, 81.604, -0.577, 56.917, -37.953, -20.502]
  Set speed (5.0 mm/s)
  MoveL 393 to (-35.89, 84.7, 119.77) mm, rotated rx -143.37 ry 0 rz -156.54 deg; joints [13.125, -50.686, 82.981, -0.338, 56.917, -38.545, -21.244]
  Set speed (16.7 mm/s)
  MoveL 394 to (-31.63, 85.22, 120.6) mm, rotated rx -143.89 ry 0 rz -159.13 deg; joints [13.217, -50.781, 83.179, -0.308, 56.917, -38.985, -18.758]
  MoveL 395 to (-31.47, 85.24, 120.63) mm, rotated rx -143.91 ry 0 rz -159.23 deg; joints [13.221, -50.785, 83.186, -0.307, 56.917, -39.002, -18.665]
  MoveL 396 to (-31.25, 85.28, 120.66) mm, rotated rx -143.95 ry 0 rz -159.48 deg; joints [13.227, -50.799, 83.196, -0.307, 56.921, -39.034, -18.415]
  MoveL 397 to (-35.37, 96.3, 136.83) mm, rotated rx -143.95 ry 0 rz -159.48 deg; joints [13.698, -50.136, 81.83, -0.543, 56.921, -38.438, -17.682]
  Set speed (1000.0 mm/s)
  MoveL 398 to (-28.57, 94.12, 139.9) mm, rotated rx -145.73 ry 0 rz -163.14 deg; joints [14.026, -50.517, 82.554, -0.439, 56.921, -39.945, -14.371]
  Set speed (5.0 mm/s)
  MoveL 399 to (-25.31, 83.34, 123.38) mm, rotated rx -145.73 ry 0 rz -163.14 deg; joints [13.54, -51.172, 83.884, -0.211, 56.921, -40.553, -15.074]
  Set speed (16.7 mm/s)
  MoveL 400 to (-22.08, 84.31, 123.33) mm, rotated rx -145.7 ry 0 rz -165.36 deg; joints [13.535, -51.167, 83.874, -0.212, 56.921, -40.53, -12.85]
  MoveL 401 to (-20.8, 84.38, 123.51) mm, rotated rx -145.7 ry 0 rz -165.36 deg; joints [13.539, -51.109, 83.891, -0.188, 56.921, -40.539, -12.928]
  MoveL 402 to (-19.95, 84.08, 123.85) mm, rotated rx -145.7 ry 0 rz -165.36 deg; joints [13.552, -51.086, 83.926, -0.17, 56.92, -40.536, -12.988]
  MoveL 403 to (-19.21, 83.3, 124.5) mm, rotated rx -145.7 ry 0 rz -165.36 deg; joints [13.579, -51.091, 83.991, -0.15, 56.92, -40.519, -13.051]
  MoveL 404 to (-19.04, 82.27, 125.2) mm, rotated rx -145.7 ry 0 rz -165.36 deg; joints [13.61, -51.131, 84.062, -0.14, 56.921, -40.493, -13.082]
  MoveL 405 to (-19.14, 81.57, 125.65) mm, rotated rx -146.01 ry 0 rz -165.18 deg; joints [13.662, -51.191, 84.183, -0.121, 56.921, -40.757, -13.332]
  MoveL 406 to (-19.61, 80.53, 126.25) mm, rotated rx -146.01 ry 0 rz -165.18 deg; joints [13.691, -51.256, 84.239, -0.121, 56.929, -40.729, -13.332]
  MoveL 407 to (-20.6, 79.78, 126.57) mm, rotated rx -146.01 ry 0 rz -165.18 deg; joints [13.706, -51.312, 84.248, -0.121, 56.977, -40.714, -13.332]
  MoveL 408 to (-24.91, 77.66, 127.1) mm, rotated rx -146.38 ry 0 rz -161.87 deg; joints [13.77, -51.387, 84.398, -0.096, 56.977, -41.038, -16.72]
  MoveL 409 to (-24.9, 77.68, 127.09) mm, rotated rx -146.75 ry 0 rz -160.82 deg; joints [13.805, -51.354, 84.492, -0.055, 56.977, -41.393, -17.901]
  MoveL 410 to (-25.42, 76.36, 127.79) mm, rotated rx -147.25 ry 0 rz -160.15 deg; joints [13.889, -51.454, 84.691, -0.022, 56.977, -41.822, -18.674]
  MoveL 411 to (-25.89, 75.63, 128.13) mm, rotated rx -147.41 ry 0 rz -159.78 deg; joints [13.922, -51.502, 84.769, -0.012, 56.977, -41.956, -19.071]
  MoveL 412 to (-26.43, 74.54, 128.65) mm, rotated rx -147.79 ry 0 rz -159.13 deg; joints [13.986, -51.581, 84.925, 0.013, 56.977, -42.289, -19.797]
  MoveL 413 to (-25.86, 74.27, 128.93) mm, rotated rx -149.16 ry 0 rz -159.29 deg; joints [14.141, -51.765, 85.306, 0.081, 56.977, -43.538, -19.847]
  MoveL 414 to (-24.57, 73.46, 129.64) mm, rotated rx -149.67 ry 0 rz -159.96 deg; joints [14.226, -51.876, 85.521, 0.116, 56.977, -43.986, -19.284]
  MoveL 415 to (-24.22, 73.63, 129.61) mm, rotated rx -150.07 ry 0 rz -161.91 deg; joints [14.268, -52.01, 85.577, 0.117, 57.054, -44.341, -17.334]
  MoveL 416 to (-23.88, 73.76, 129.6) mm, rotated rx -150.06 ry 0 rz -162.18 deg; joints [14.267, -52.008, 85.574, 0.116, 57.054, -44.334, -17.066]
  MoveL 417 to (-22.47, 74.19, 129.6) mm, rotated rx -150.06 ry 0 rz -163.14 deg; joints [14.267, -52, 85.575, 0.119, 57.054, -44.339, -16.111]
  MoveL 418 to (-22.37, 74.86, 129.24) mm, rotated rx -149.32 ry 0 rz -164.96 deg; joints [14.181, -51.995, 85.341, 0.041, 57.054, -43.642, -14.057]
  MoveL 419 to (-22.31, 75.05, 129.14) mm, rotated rx -149.25 ry 0 rz -165.04 deg; joints [14.169, -51.98, 85.311, 0.036, 57.054, -43.579, -13.962]
  MoveL 420 to (-22.08, 75.53, 128.9) mm, rotated rx -149.25 ry 0 rz -165.04 deg; joints [14.157, -51.949, 85.286, 0.036, 57.048, -43.591, -13.962]
  MoveL 421 to (-21.38, 76.61, 128.38) mm, rotated rx -148.88 ry 0 rz -165.71 deg; joints [14.094, -51.869, 85.131, 0.011, 57.048, -43.266, -13.207]
  MoveL 422 to (-21.39, 76.6, 128.38) mm, rotated rx -148.51 ry 0 rz -166.12 deg; joints [14.058, -51.852, 85.038, -0.015, 57.048, -42.92, -12.724]
  MoveL 423 to (-21.22, 78.23, 127.43) mm, rotated rx -147.83 ry 0 rz -166.52 deg; joints [13.944, -51.71, 84.761, -0.06, 57.048, -42.333, -12.187]
  MoveL 424 to (-20.87, 79.14, 126.92) mm, rotated rx -147.83 ry 0 rz -166.52 deg; joints [13.919, -51.654, 84.707, -0.06, 57.046, -42.357, -12.187]
  MoveL 425 to (-20.67, 79.44, 126.76) mm, rotated rx -147.72 ry 0 rz -166.7 deg; joints [13.901, -51.632, 84.664, -0.067, 57.046, -42.265, -11.98]
  MoveL 426 to (-19.98, 80.12, 126.45) mm, rotated rx -147.72 ry 0 rz -166.7 deg; joints [13.886, -51.584, 84.644, -0.067, 57.017, -42.28, -11.98]
  MoveL 427 to (-17.08, 81.97, 125.69) mm, rotated rx -147.2 ry 0 rz -168.92 deg; joints [13.796, -51.476, 84.433, -0.101, 57.017, -41.828, -9.656]
  MoveL 428 to (-17.09, 81.98, 125.67) mm, rotated rx -145.8 ry 0 rz -169.64 deg; joints [13.649, -51.358, 84.083, -0.175, 57.018, -40.531, -8.696]
  MoveL 429 to (-18.66, 83.27, 124.6) mm, rotated rx -145.06 ry 0 rz -168.75 deg; joints [13.522, -51.214, 83.794, -0.221, 57.018, -39.899, -9.437]
  MoveL 430 to (-20.89, 94.5, 141) mm, rotated rx -145.06 ry 0 rz -168.75 deg; joints [14.003, -50.552, 82.452, -0.451, 57.018, -39.297, -8.727]
  Set speed (1000.0 mm/s)
  MoveL 431 to (-18.77, 98.7, 138.4) mm, rotated rx -144.84 ry 0 rz -168.92 deg; joints [13.858, -50.264, 82.141, -0.455, 57.018, -39.218, -8.53]
  Set speed (5.0 mm/s)
  MoveL 432 to (-16.55, 87.4, 122.05) mm, rotated rx -144.84 ry 0 rz -168.92 deg; joints [13.379, -50.924, 83.491, -0.224, 57.018, -39.819, -9.248]
  Set speed (16.7 mm/s)
  MoveL 433 to (-13.72, 87.38, 122.4) mm, rotated rx -145.07 ry 0 rz -170.72 deg; joints [13.419, -50.969, 83.581, -0.21, 57.018, -40.017, -7.499]
  MoveL 434 to (-13.64, 87.42, 122.39) mm, rotated rx -145.08 ry 0 rz -171.35 deg; joints [13.422, -51.016, 83.581, -0.225, 57.018, -40.012, -6.818]
  MoveL 435 to (-9.28, 88.48, 122.04) mm, rotated rx -144.85 ry 0 rz -174.23 deg; joints [13.382, -50.972, 83.492, -0.239, 57.018, -39.816, -3.89]
  MoveL 436 to (-10.44, 99.93, 138.39) mm, rotated rx -144.85 ry 0 rz -174.23 deg; joints [13.861, -50.313, 82.143, -0.47, 57.018, -39.215, -3.173]
  Set speed (1000.0 mm/s)
  MoveL 437 to (-7.68, 99.26, 139.05) mm, rotated rx -145.21 ry 0 rz -175.95 deg; joints [13.929, -50.401, 82.294, -0.452, 57.018, -39.515, -1.52]
  Set speed (5.0 mm/s)
  MoveL 438 to (-6.88, 87.88, 122.63) mm, rotated rx -145.21 ry 0 rz -175.95 deg; joints [13.448, -51.06, 83.635, -0.222, 57.018, -40.118, -2.231]
  Set speed (16.7 mm/s)
  MoveL 439 to (-6.64, 87.94, 122.59) mm, rotated rx -145.2 ry 0 rz -176 deg; joints [13.445, -51.051, 83.633, -0.221, 57.013, -40.113, -2.181]
  MoveL 440 to (-5.17, 88.26, 122.44) mm, rotated rx -145.03 ry 0 rz -177.34 deg; joints [13.421, -51.054, 83.576, -0.24, 57.013, -39.955, -0.778]
  MoveL 441 to (-2.33, 90.05, 121.22) mm, rotated rx -144.16 ry 0 rz -179.45 deg; joints [13.275, -50.916, 83.252, -0.297, 57.013, -39.199, 1.52]
  MoveL 442 to (-1.85, 90.27, 121.06) mm, rotated rx -144.16 ry 0 rz -179.45 deg; joints [13.268, -50.892, 83.246, -0.298, 56.994, -39.207, 1.521]
  MoveL 443 to (-1.69, 90.33, 121.02) mm, rotated rx -144.13 ry 0 rz -179.55 deg; joints [13.263, -50.887, 83.236, -0.299, 56.995, -39.185, 1.628]
  MoveL 444 to (-1.28, 90.44, 120.94) mm, rotated rx -144.13 ry 0 rz -179.55 deg; joints [13.259, -50.868, 83.236, -0.298, 56.98, -39.189, 1.624]
  MoveL 445 to (-0.56, 90.58, 120.84) mm, rotated rx -144.08 ry 0 rz 180 deg; joints [13.249, -50.858, 83.215, -0.301, 56.98, -39.147, 2.086]
  MoveL 446 to (-0.09, 90.65, 120.79) mm, rotated rx -143.97 ry 0 rz 179.38 deg; joints [13.237, -50.871, 83.185, -0.314, 56.98, -39.045, 2.751]
  MoveL 447 to (0.17, 90.74, 120.72) mm, rotated rx -143.93 ry 0 rz 179.22 deg; joints [13.229, -50.862, 83.168, -0.317, 56.98, -39.007, 2.919]
  MoveL 448 to (3.8, 92.42, 119.38) mm, rotated rx -143.04 ry 0 rz 176.83 deg; joints [13.075, -50.715, 82.837, -0.372, 56.979, -38.243, 5.498]
  MoveL 449 to (4.11, 92.58, 119.25) mm, rotated rx -142.93 ry 0 rz 176.57 deg; joints [13.057, -50.704, 82.8, -0.379, 56.979, -38.146, 5.788]
  MoveL 450 to (7.34, 94.25, 117.77) mm, rotated rx -142 ry 0 rz 174.62 deg; joints [12.891, -50.544, 82.454, -0.433, 56.979, -37.352, 7.929]
  MoveL 451 to (7.29, 94.23, 117.79) mm, rotated rx -141.72 ry 0 rz 174.25 deg; joints [12.863, -50.55, 82.393, -0.453, 56.979, -37.09, 8.371]
  MoveL 452 to (8, 95.05, 117.08) mm, rotated rx -141.29 ry 0 rz 173.87 deg; joints [12.785, -50.476, 82.236, -0.476, 56.979, -36.732, 8.827]
  MoveL 453 to (7.98, 95.04, 117.09) mm, rotated rx -140.27 ry 0 rz 174.01 deg; joints [12.668, -50.354, 82.001, -0.507, 56.979, -35.806, 8.809]
  MoveL 454 to (7.61, 95.5, 116.74) mm, rotated rx -140.06 ry 0 rz 174.26 deg; joints [12.63, -50.319, 81.925, -0.518, 56.979, -35.63, 8.603]
  MoveL 455 to (8.89, 108.27, 132.08) mm, rotated rx -140.06 ry 0 rz 174.26 deg; joints [13.07, -49.643, 80.489, -0.768, 56.979, -35.061, 9.394]
  Set speed (1000.0 mm/s)
  MoveL 456 to (6.54, 110.49, 130.37) mm, rotated rx -139 ry 0 rz 175.84 deg; joints [12.877, -49.447, 80.112, -0.814, 56.979, -34.173, 7.992]
  Set speed (5.0 mm/s)
  MoveL 457 to (5.59, 97.4, 115.28) mm, rotated rx -139 ry 0 rz 175.84 deg; joints [12.446, -50.126, 81.568, -0.561, 56.979, -34.734, 7.184]
  Set speed (16.7 mm/s)
  MoveL 458 to (1.93, 99.67, 113.44) mm, rotated rx -137.93 ry 0 rz 178.05 deg; joints [12.246, -49.95, 81.189, -0.613, 56.979, -33.835, 5.187]
  MoveL 459 to (-0.96, 100.61, 112.62) mm, rotated rx -137.37 ry 0 rz -180 deg; joints [12.146, -49.838, 81.005, -0.63, 56.979, -33.372, 3.308]
  MoveL 460 to (-1.57, 100.68, 112.55) mm, rotated rx -137.27 ry 0 rz -179.5 deg; joints [12.13, -49.812, 80.978, -0.63, 56.977, -33.286, 2.814]
  MoveL 461 to (-4.78, 101.28, 111.93) mm, rotated rx -136.92 ry 0 rz -177.69 deg; joints [12.063, -49.756, 80.855, -0.646, 56.977, -32.989, 1.064]
  MoveL 462 to (-5.33, 114.93, 126.53) mm, rotated rx -136.92 ry 0 rz -177.69 deg; joints [12.477, -49.073, 79.362, -0.905, 56.977, -32.444, 1.905]
  Set speed (1000.0 mm/s)
  MoveL 463 to (-6.43, 118.47, 123.16) mm, rotated rx -136.55 ry 0 rz -177.89 deg; joints [12.304, -49.012, 79.049, -0.969, 56.977, -32.217, 2.367]
  Set speed (5.0 mm/s)
  MoveL 464 to (-5.93, 104.72, 108.65) mm, rotated rx -136.55 ry 0 rz -177.89 deg; joints [11.893, -49.691, 80.546, -0.709, 56.977, -32.759, 1.518]
  Set speed (16.7 mm/s)
  MoveL 465 to (-5.24, 105.5, 107.92) mm, rotated rx -136.16 ry 0 rz -178.28 deg; joints [11.818, -49.632, 80.415, -0.725, 56.977, -32.436, 1.978]
  MoveL 466 to (-5.13, 105.96, 107.49) mm, rotated rx -135.65 ry 0 rz -178.52 deg; joints [11.741, -49.59, 80.279, -0.748, 56.977, -31.993, 2.319]
  MoveL 467 to (-4.87, 106.64, 106.81) mm, rotated rx -135.29 ry 0 rz -178.67 deg; joints [11.672, -49.537, 80.16, -0.763, 56.977, -31.696, 2.536]
  MoveL 468 to (-4.79, 106.65, 106.82) mm, rotated rx -134.3 ry 0 rz -176.56 deg; joints [11.546, -49.284, 80.007, -0.763, 56.859, -30.826, 0.443]
  MoveL 469 to (-5.42, 106.22, 107.21) mm, rotated rx -134.51 ry 0 rz -176.21 deg; joints [11.587, -49.315, 80.076, -0.754, 56.859, -31.002, 0.053]
  MoveL 470 to (-5.39, 106.23, 107.2) mm, rotated rx -134.97 ry 0 rz -175.8 deg; joints [11.64, -49.313, 80.168, -0.731, 56.859, -31.419, -0.452]
  MoveL 471 to (-5.89, 104.67, 108.71) mm, rotated rx -135.79 ry 0 rz -175.47 deg; joints [11.797, -49.434, 80.441, -0.696, 56.859, -32.099, -0.941]
  MoveL 472 to (-6.99, 118.57, 123.04) mm, rotated rx -135.79 ry 0 rz -175.47 deg; joints [12.201, -48.751, 78.927, -0.958, 56.859, -31.562, -0.079]
  Set speed (1000.0 mm/s)
  MoveL 473 to (-9.78, 115.15, 126.06) mm, rotated rx -136.65 ry 0 rz -175.11 deg; joints [12.43, -49.053, 79.332, -0.942, 56.859, -32.205, -0.536]
  Set speed (5.0 mm/s)
  MoveL 474 to (-8.61, 101.47, 111.52) mm, rotated rx -136.65 ry 0 rz -175.11 deg; joints [12.019, -49.735, 80.829, -0.681, 56.859, -32.749, -1.381]
  Set speed (16.7 mm/s)
  MoveL 475 to (-9.21, 101.41, 111.53) mm, rotated rx -136.66 ry 0 rz -174.77 deg; joints [12.02, -49.736, 80.831, -0.681, 56.859, -32.754, -1.721]
  MoveL 476 to (-9.17, 101.41, 111.53) mm, rotated rx -136.98 ry 0 rz -173.78 deg; joints [12.054, -49.668, 80.898, -0.643, 56.859, -33.067, -2.856]
  MoveL 477 to (-11.88, 98.43, 113.91) mm, rotated rx -138.36 ry 0 rz -172.02 deg; joints [12.311, -49.885, 81.376, -0.577, 56.859, -34.214, -4.883]
  MoveL 478 to (-14.94, 94.64, 116.73) mm, rotated rx -140.02 ry 0 rz -169.88 deg; joints [12.62, -50.16, 81.974, -0.492, 56.859, -35.619, -7.355]
  MoveL 479 to (-14.92, 94.66, 116.72) mm, rotated rx -140.72 ry 0 rz -169.55 deg; joints [12.697, -50.204, 82.13, -0.46, 56.859, -36.252, -7.793]
  MoveL 480 to (-14.63, 93.76, 117.48) mm, rotated rx -141.18 ry 0 rz -169.63 deg; joints [12.781, -50.283, 82.299, -0.435, 56.859, -36.64, -7.811]
  MoveL 481 to (-14.58, 93.06, 118.04) mm, rotated rx -141.18 ry 0 rz -169.63 deg; joints [12.804, -50.309, 82.346, -0.429, 56.859, -36.619, -7.833]
  MoveL 482 to (-14.62, 92.8, 118.24) mm, rotated rx -141.3 ry 0 rz -169.58 deg; joints [12.827, -50.331, 82.391, -0.422, 56.859, -36.722, -7.909]
  MoveL 483 to (-14.7, 92.49, 118.48) mm, rotated rx -141.3 ry 0 rz -169.58 deg; joints [12.837, -50.347, 82.412, -0.422, 56.859, -36.712, -7.913]
  MoveL 484 to (-15.55, 89.92, 120.33) mm, rotated rx -142.45 ry 0 rz -168.75 deg; joints [13.045, -50.553, 82.844, -0.356, 56.859, -37.694, -8.972]
  MoveL 485 to (-16.23, 88.97, 120.95) mm, rotated rx -142.7 ry 0 rz -168.34 deg; joints [13.099, -50.619, 82.958, -0.342, 56.859, -37.894, -9.433]
  MoveL 486 to (-17.08, 87.31, 122.03) mm, rotated rx -143.4 ry 0 rz -167.58 deg; joints [13.224, -50.748, 83.225, -0.301, 56.859, -38.492, -10.336]
  MoveL 487 to (-19.65, 98.95, 138.09) mm, rotated rx -143.4 ry 0 rz -167.58 deg; joints [13.691, -50.081, 81.847, -0.539, 56.859, -37.9, -9.596]
  Set speed (1000.0 mm/s)
  MoveL 488 to (-23.25, 95.87, 139.7) mm, rotated rx -143.97 ry 0 rz -166.76 deg; joints [13.83, -50.362, 82.133, -0.539, 56.867, -38.325, -10.431]
  Set speed (5.0 mm/s)
  MoveL 489 to (-20.56, 84.42, 123.52) mm, rotated rx -143.97 ry 0 rz -166.76 deg; joints [13.359, -51.027, 83.497, -0.303, 56.867, -38.921, -11.159]
  Set speed (16.7 mm/s)
  MoveL 490 to (-23.6, 84.33, 123.04) mm, rotated rx -143.65 ry 0 rz -164.8 deg; joints [13.302, -50.967, 83.374, -0.322, 56.867, -38.648, -13.05]
  MoveL 491 to (-23.58, 84.33, 123.04) mm, rotated rx -143.67 ry 0 rz -163.84 deg; joints [13.3, -50.889, 83.378, -0.296, 56.867, -38.683, -14.089]
  MoveL 492 to (-24.36, 83.85, 123.22) mm, rotated rx -143.78 ry 0 rz -163.26 deg; joints [13.321, -50.911, 83.424, -0.289, 56.867, -38.785, -14.695]
  MoveL 493 to (-27.76, 95.16, 139.36) mm, rotated rx -143.78 ry 0 rz -163.26 deg; joints [13.791, -50.245, 82.055, -0.526, 56.867, -38.19, -13.963]
  Set speed (1000.0 mm/s)
  MoveL 494 to (-35.24, 96.75, 136.54) mm, rotated rx -142.35 ry 0 rz -160.89 deg; joints [13.519, -50.096, 81.457, -0.662, 56.867, -36.953, -15.872]
  Set speed (5.0 mm/s)
  MoveL 495 to (-31.24, 85.21, 120.71) mm, rotated rx -142.35 ry 0 rz -160.89 deg; joints [13.06, -50.765, 82.851, -0.418, 56.867, -37.539, -16.627]
  Set speed (16.7 mm/s)
  MoveL 496 to (-31.61, 85.31, 120.54) mm, rotated rx -142.24 ry 0 rz -160.69 deg; joints [13.041, -50.746, 82.811, -0.424, 56.867, -37.449, -16.806]
  MoveL 497 to (-32.59, 85.86, 119.89) mm, rotated rx -142.24 ry 0 rz -160.69 deg; joints [13.016, -50.759, 82.754, -0.445, 56.867, -37.464, -16.735]
  MoveL 498 to (-33.02, 86.8, 119.09) mm, rotated rx -142.24 ry 0 rz -160.69 deg; joints [12.983, -50.731, 82.685, -0.457, 56.867, -37.491, -16.692]
  MoveL 499 to (-33.05, 87.15, 118.83) mm, rotated rx -142.08 ry 0 rz -160.74 deg; joints [12.953, -50.702, 82.624, -0.466, 56.867, -37.353, -16.609]
  MoveL 500 to (-33.06, 87.43, 118.62) mm, rotated rx -142.08 ry 0 rz -160.74 deg; joints [12.944, -50.688, 82.606, -0.467, 56.867, -37.361, -16.604]
  MoveL 501 to (-32.96, 88.58, 117.78) mm, rotated rx -141.57 ry 0 rz -161.02 deg; joints [12.853, -50.599, 82.418, -0.495, 56.867, -36.935, -16.224]
  MoveL 502 to (-32.9, 88.59, 117.79) mm, rotated rx -140.37 ry 0 rz -159.14 deg; joints [12.708, -50.313, 82.155, -0.495, 56.831, -35.871, -18.094]
  MoveL 503 to (-33.33, 88.3, 117.9) mm, rotated rx -140.55 ry 0 rz -158.45 deg; joints [12.731, -50.302, 82.204, -0.477, 56.831, -36.04, -18.847]
  MoveL 504 to (-33.48, 88.12, 117.99) mm, rotated rx -140.6 ry 0 rz -158.32 deg; joints [12.741, -50.311, 82.224, -0.474, 56.831, -36.086, -18.98]
  MoveL 505 to (-35.76, 84.84, 119.71) mm, rotated rx -141.71 ry 0 rz -156.15 deg; joints [12.938, -50.495, 82.628, -0.412, 56.831, -37.027, -21.377]
  MoveL 506 to (-40.77, 96.17, 135.41) mm, rotated rx -141.71 ry 0 rz -156.15 deg; joints [13.391, -49.823, 81.219, -0.657, 56.831, -36.445, -20.61]
  Set speed (1000.0 mm/s)
  MoveL 507 to (-45.17, 95.45, 134.52) mm, rotated rx -141.64 ry 0 rz -155.98 deg; joints [13.359, -49.999, 81.136, -0.738, 56.831, -36.366, -20.517]
  Set speed (5.0 mm/s)
  MoveL 508 to (-40.11, 84.12, 118.84) mm, rotated rx -141.64 ry 0 rz -155.98 deg; joints [12.906, -50.668, 82.541, -0.491, 56.831, -36.947, -21.283]
  Set speed (16.7 mm/s)
  MoveL 509 to (-43.3, 87.22, 115.43) mm, rotated rx -139.58 ry 0 rz -155 deg; joints [12.529, -50.315, 81.789, -0.599, 56.831, -35.208, -21.85]
  MoveL 510 to (-43.57, 87.55, 115.08) mm, rotated rx -139.58 ry 0 rz -155 deg; joints [12.515, -50.307, 81.762, -0.605, 56.831, -35.219, -21.829]
  MoveL 511 to (-43.75, 87.84, 114.79) mm, rotated rx -139.41 ry 0 rz -154.98 deg; joints [12.484, -50.279, 81.701, -0.613, 56.831, -35.077, -21.816]
  MoveL 512 to (-43.84, 88.04, 114.6) mm, rotated rx -139.41 ry 0 rz -154.98 deg; joints [12.476, -50.273, 81.686, -0.615, 56.831, -35.084, -21.808]
  MoveL 513 to (-44.64, 90.03, 112.73) mm, rotated rx -138.33 ry 0 rz -155.05 deg; joints [12.275, -50.098, 81.306, -0.668, 56.831, -34.183, -21.53]
  MoveL 514 to (-44.6, 90.01, 112.76) mm, rotated rx -137.53 ry 0 rz -154.46 deg; joints [12.179, -49.961, 81.13, -0.675, 56.831, -33.474, -22.08]
  MoveL 515 to (-47.82, 90.06, 111.4) mm, rotated rx -136.76 ry 0 rz -152.84 deg; joints [12.033, -49.838, 80.862, -0.71, 56.831, -32.826, -23.556]
  MoveL 516 to (-48.39, 90.12, 111.1) mm, rotated rx -136.76 ry 0 rz -152.84 deg; joints [12.022, -49.855, 80.842, -0.72, 56.831, -32.831, -23.518]
  MoveL 517 to (-48.53, 90.16, 111.01) mm, rotated rx -136.71 ry 0 rz -152.78 deg; joints [12.013, -49.848, 80.825, -0.723, 56.831, -32.79, -23.569]
  MoveL 518 to (-49.07, 90.37, 110.6) mm, rotated rx -136.71 ry 0 rz -152.78 deg; joints [11.997, -49.855, 80.797, -0.732, 56.831, -32.801, -23.532]
  MoveL 519 to (-50.17, 91.04, 109.55) mm, rotated rx -136.12 ry 0 rz -152.4 deg; joints [11.886, -49.767, 80.599, -0.758, 56.83, -32.314, -23.798]
  MoveL 520 to (-50.02, 90.97, 109.68) mm, rotated rx -136.01 ry 0 rz -152.3 deg; joints [11.877, -49.749, 80.587, -0.758, 56.822, -32.211, -23.891]
  MoveL 521 to (-51.81, 91.46, 108.44) mm, rotated rx -135.32 ry 0 rz -151.55 deg; joints [11.745, -49.645, 80.357, -0.787, 56.822, -31.637, -24.518]
  MoveL 522 to (-52.18, 91.59, 108.14) mm, rotated rx -135.32 ry 0 rz -151.55 deg; joints [11.734, -49.651, 80.338, -0.793, 56.822, -31.645, -24.493]
  MoveL 523 to (-52.78, 92.16, 107.37) mm, rotated rx -135.32 ry 0 rz -151.55 deg; joints [11.705, -49.642, 80.287, -0.804, 56.822, -31.669, -24.449]
  MoveL 524 to (-53.01, 92.57, 106.9) mm, rotated rx -135.07 ry 0 rz -151.55 deg; joints [11.656, -49.605, 80.204, -0.814, 56.822, -31.46, -24.403]
  MoveL 525 to (-53.17, 93.2, 106.27) mm, rotated rx -135.07 ry 0 rz -151.55 deg; joints [11.631, -49.578, 80.161, -0.817, 56.822, -31.484, -24.387]
  MoveL 526 to (-53.1, 96.96, 102.89) mm, rotated rx -133.3 ry 0 rz -152.5 deg; joints [11.285, -49.327, 79.588, -0.884, 56.822, -30.026, -23.111]
  MoveL 527 to (-52.96, 97.63, 102.33) mm, rotated rx -131.79 ry 0 rz -152.04 deg; joints [11.074, -49.111, 79.254, -0.902, 56.821, -28.72, -23.449]
  MoveL 528 to (-54.46, 97.31, 101.85) mm, rotated rx -131.54 ry 0 rz -151.28 deg; joints [11.025, -49.078, 79.177, -0.911, 56.821, -28.516, -24.167]
  MoveL 529 to (-55.01, 97.23, 101.62) mm, rotated rx -131.54 ry 0 rz -151.28 deg; joints [11.017, -49.101, 79.165, -0.92, 56.822, -28.519, -24.132]
  MoveL 530 to (-56.07, 97.47, 100.81) mm, rotated rx -131.54 ry 0 rz -151.28 deg; joints [10.989, -49.127, 79.122, -0.936, 56.822, -28.539, -24.061]
  MoveL 531 to (-56.25, 97.58, 100.61) mm, rotated rx -131.44 ry 0 rz -151.22 deg; joints [10.968, -49.113, 79.09, -0.939, 56.822, -28.455, -24.096]
  MoveL 532 to (-56.8, 98.31, 99.58) mm, rotated rx -131.44 ry 0 rz -151.22 deg; joints [10.93, -49.095, 79.031, -0.947, 56.821, -28.49, -24.055]
  MoveL 533 to (-57.06, 99.51, 98.22) mm, rotated rx -130.76 ry 0 rz -151.4 deg; joints [10.794, -49.009, 78.827, -0.969, 56.821, -27.939, -23.764]
  MoveL 534 to (-57.33, 99.74, 97.84) mm, rotated rx -130.61 ry 0 rz -151.38 deg; joints [10.761, -48.993, 78.778, -0.975, 56.821, -27.818, -23.747]
  MoveL 535 to (-57.59, 100.47, 96.93) mm, rotated rx -130.27 ry 0 rz -151.34 deg; joints [10.684, -48.934, 78.662, -0.983, 56.821, -27.549, -23.73]
  MoveL 536 to (-57.51, 102.68, 94.63) mm, rotated rx -129.14 ry 0 rz -151.89 deg; joints [10.456, -48.797, 78.334, -1.015, 56.821, -26.638, -22.99]
  MoveL 537 to (-64.82, 116.37, 107.26) mm, rotated rx -129.14 ry 0 rz -151.89 deg; joints [10.805, -48.115, 76.725, -1.284, 56.821, -26.159, -22.034]
  Set speed (1000.0 mm/s)
  MoveL 538 to (-61.57, 118.93, 106.35) mm, rotated rx -129.16 ry 0 rz -152.04 deg; joints [10.767, -47.953, 76.725, -1.273, 56.697, -26.213, -21.916]
  Set speed (5.0 mm/s)
  MoveL 539 to (-54.3, 105.24, 93.72) mm, rotated rx -129.16 ry 0 rz -152.04 deg; joints [10.419, -48.634, 78.338, -1.003, 56.697, -26.693, -22.876]
  Set speed (16.7 mm/s)
  MoveL 540 to (-52.25, 105.41, 94.68) mm, rotated rx -129.62 ry 0 rz -152.96 deg; joints [10.513, -48.69, 78.473, -0.99, 56.697, -27.07, -22.038]
  MoveL 541 to (-52.32, 105.39, 94.67) mm, rotated rx -129.76 ry 0 rz -153.46 deg; joints [10.531, -48.737, 78.476, -0.99, 56.744, -27.193, -21.54]
  MoveL 542 to (-50.68, 106.06, 94.82) mm, rotated rx -129.84 ry 0 rz -154.32 deg; joints [10.546, -48.745, 78.497, -0.988, 56.744, -27.253, -20.692]
  MoveL 543 to (-50.29, 106.19, 94.87) mm, rotated rx -129.85 ry 0 rz -154.43 deg; joints [10.55, -48.737, 78.502, -0.984, 56.744, -27.266, -20.6]
  MoveL 544 to (-48.62, 106.73, 95.14) mm, rotated rx -129.99 ry 0 rz -155.41 deg; joints [10.579, -48.769, 78.544, -0.984, 56.744, -27.382, -19.633]
  MoveL 545 to (-48.14, 106.92, 95.18) mm, rotated rx -130.01 ry 0 rz -155.66 deg; joints [10.582, -48.771, 78.549, -0.984, 56.744, -27.395, -19.383]
  MoveL 546 to (-44.06, 108.2, 95.7) mm, rotated rx -130.26 ry 0 rz -157.64 deg; joints [10.632, -48.79, 78.622, -0.974, 56.744, -27.599, -17.455]
  MoveL 547 to (-42.82, 108.32, 96.12) mm, rotated rx -130.26 ry 0 rz -157.64 deg; joints [10.645, -48.732, 78.64, -0.955, 56.744, -27.596, -17.533]
  MoveL 548 to (-42.06, 108.1, 96.71) mm, rotated rx -130.26 ry 0 rz -157.64 deg; joints [10.665, -48.711, 78.67, -0.943, 56.744, -27.581, -17.584]
  MoveL 549 to (-41.68, 107.78, 97.23) mm, rotated rx -130.26 ry 0 rz -157.64 deg; joints [10.684, -48.71, 78.698, -0.937, 56.744, -27.565, -17.614]
  MoveL 550 to (-41.44, 107.16, 98.02) mm, rotated rx -130.26 ry 0 rz -157.64 deg; joints [10.714, -48.73, 78.742, -0.933, 56.744, -27.538, -17.639]
  MoveL 551 to (-41.61, 106.43, 98.74) mm, rotated rx -130.26 ry 0 rz -157.64 deg; joints [10.742, -48.766, 78.779, -0.932, 56.754, -27.51, -17.649]
  MoveL 552 to (-41.91, 105.85, 99.24) mm, rotated rx -130.51 ry 0 rz -157.39 deg; joints [10.792, -48.798, 78.854, -0.924, 56.754, -27.716, -17.942]
  MoveL 553 to (-42.02, 105.65, 99.4) mm, rotated rx -130.51 ry 0 rz -157.39 deg; joints [10.799, -48.809, 78.861, -0.924, 56.76, -27.71, -17.944]
  MoveL 554 to (-42.66, 104.64, 100.19) mm, rotated rx -130.92 ry 0 rz -156.89 deg; joints [10.879, -48.86, 78.982, -0.911, 56.76, -28.038, -18.514]
  MoveL 555 to (-42.71, 104.67, 100.13) mm, rotated rx -132.48 ry 0 rz -157.93 deg; joints [11.076, -49.101, 79.285, -0.909, 56.76, -29.403, -17.542]
  MoveL 556 to (-42.56, 104.75, 100.12) mm, rotated rx -132.47 ry 0 rz -157.99 deg; joints [11.075, -49.099, 79.284, -0.909, 56.758, -29.4, -17.479]
  MoveL 557 to (-40.52, 105.67, 99.99) mm, rotated rx -132.41 ry 0 rz -159.12 deg; joints [11.061, -49.09, 79.264, -0.911, 56.758, -29.345, -16.334]
  MoveL 558 to (-45.78, 119.47, 113.47) mm, rotated rx -132.41 ry 0 rz -159.12 deg; joints [11.438, -48.41, 77.7, -1.179, 56.759, -28.836, -15.42]
  Set speed (1000.0 mm/s)
  MoveL 559 to (-43.02, 122.52, 111.29) mm, rotated rx -131.42 ry 0 rz -160.42 deg; joints [11.232, -48.24, 77.38, -1.202, 56.759, -28.042, -13.974]
  Set speed (5.0 mm/s)
  MoveL 560 to (-38, 108.39, 98.06) mm, rotated rx -131.42 ry 0 rz -160.42 deg; joints [10.864, -48.921, 78.96, -0.933, 56.759, -28.543, -14.903]
  Set speed (16.7 mm/s)
  MoveL 561 to (-35.84, 108.8, 98.41) mm, rotated rx -131.59 ry 0 rz -161.5 deg; joints [10.899, -48.944, 79.013, -0.927, 56.759, -28.687, -13.85]
  MoveL 562 to (-35.69, 108.96, 98.29) mm, rotated rx -131.11 ry 0 rz -162.92 deg; joints [10.843, -49.053, 78.929, -0.974, 56.759, -28.24, -12.23]
  MoveL 563 to (-35.48, 109.37, 97.91) mm, rotated rx -130.92 ry 0 rz -163.08 deg; joints [10.804, -49.029, 78.871, -0.98, 56.759, -28.085, -12.039]
  MoveL 564 to (-34.6, 111.34, 95.99) mm, rotated rx -129.93 ry 0 rz -163.81 deg; joints [10.609, -48.911, 78.583, -1.009, 56.759, -27.278, -11.142]
  MoveL 565 to (-36.6, 110.9, 95.75) mm, rotated rx -128.56 ry 0 rz -161.05 deg; joints [10.421, -48.648, 78.354, -1.009, 56.67, -26.094, -13.844]
  MoveL 566 to (-38.39, 109.26, 96.92) mm, rotated rx -129.14 ry 0 rz -159.95 deg; joints [10.538, -48.717, 78.521, -0.993, 56.67, -26.564, -15.049]
  MoveL 567 to (-39.39, 108.62, 97.25) mm, rotated rx -129.14 ry 0 rz -159.95 deg; joints [10.552, -48.767, 78.521, -0.996, 56.712, -26.55, -15.04]
  MoveL 568 to (-40.02, 108.41, 97.23) mm, rotated rx -129.14 ry 0 rz -159.95 deg; joints [10.553, -48.802, 78.521, -1.004, 56.716, -26.545, -15.008]
  MoveL 569 to (-40.83, 108.3, 97.01) mm, rotated rx -129.14 ry 0 rz -159.95 deg; joints [10.547, -48.843, 78.513, -1.016, 56.716, -26.545, -14.959]
  MoveL 570 to (-41.87, 108.5, 96.34) mm, rotated rx -129.14 ry 0 rz -159.95 deg; joints [10.524, -48.879, 78.482, -1.031, 56.716, -26.561, -14.89]
  MoveL 571 to (-42.38, 108.74, 95.85) mm, rotated rx -128.9 ry 0 rz -159.75 deg; joints [10.475, -48.85, 78.412, -1.038, 56.716, -26.363, -15.043]
  MoveL 572 to (-42.97, 109.28, 94.96) mm, rotated rx -128.9 ry 0 rz -159.75 deg; joints [10.443, -48.852, 78.367, -1.047, 56.716, -26.391, -14.996]
  MoveL 573 to (-43.02, 110.11, 93.98) mm, rotated rx -128.9 ry 0 rz -159.75 deg; joints [10.406, -48.818, 78.315, -1.049, 56.715, -26.427, -14.977]
  MoveL 574 to (-42.61, 110.81, 93.34) mm, rotated rx -128.9 ry 0 rz -159.75 deg; joints [10.381, -48.779, 78.289, -1.049, 56.695, -26.452, -14.97]
  MoveL 575 to (-39.45, 114.19, 90.61) mm, rotated rx -127.6 ry 0 rz -161.71 deg; joints [10.115, -48.629, 77.925, -1.079, 56.695, -25.404, -12.801]
  MoveL 576 to (-38.76, 114.71, 90.25) mm, rotated rx -127.6 ry 0 rz -161.71 deg; joints [10.1, -48.594, 77.921, -1.079, 56.66, -25.418, -12.798]
  MoveL 577 to (-38.14, 115.07, 90.06) mm, rotated rx -127.51 ry 0 rz -162.04 deg; joints [10.082, -48.585, 77.897, -1.081, 56.66, -25.346, -12.449]
  MoveL 578 to (-32.45, 117.85, 88.68) mm, rotated rx -126.88 ry 0 rz -164.92 deg; joints [9.95, -48.507, 77.723, -1.093, 56.66, -24.839, -9.474]
  MoveL 579 to (-31.78, 118.21, 88.45) mm, rotated rx -126.78 ry 0 rz -165.19 deg; joints [9.929, -48.487, 77.694, -1.093, 56.66, -24.765, -9.196]
  MoveL 580 to (-27.47, 119.84, 87.7) mm, rotated rx -126.43 ry 0 rz -167.33 deg; joints [9.856, -48.449, 77.6, -1.1, 56.66, -24.482, -7.002]
  MoveL 581 to (-31, 135.54, 99.57) mm, rotated rx -126.43 ry 0 rz -167.33 deg; joints [10.181, -47.77, 75.954, -1.369, 56.66, -24.028, -6.006]
  Set speed (1000.0 mm/s)
  MoveL 582 to (-27.64, 135.23, 100.97) mm, rotated rx -126.99 ry 0 rz -168.76 deg; joints [10.303, -47.845, 76.115, -1.362, 56.66, -24.465, -4.657]
  Set speed (5.0 mm/s)
  MoveL 583 to (-24.52, 119.56, 88.93) mm, rotated rx -126.99 ry 0 rz -168.76 deg; joints [9.973, -48.524, 77.754, -1.092, 56.66, -24.925, -5.645]
  Set speed (16.7 mm/s)
  MoveL 584 to (-23.46, 119.99, 88.66) mm, rotated rx -126.85 ry 0 rz -169.29 deg; joints [9.946, -48.51, 77.718, -1.095, 56.66, -24.819, -5.096]
  MoveL 585 to (-22.96, 120.18, 88.53) mm, rotated rx -126.7 ry 0 rz -169.8 deg; joints [9.923, -48.529, 77.689, -1.104, 56.66, -24.683, -4.539]
  MoveL 586 to (-16.96, 123.4, 85.38) mm, rotated rx -125.24 ry 0 rz -172.77 deg; joints [9.621, -48.376, 77.307, -1.13, 56.66, -23.519, -1.342]
  MoveL 587 to (-16.95, 123.4, 85.38) mm, rotated rx -124.49 ry 0 rz -173.33 deg; joints [9.526, -48.399, 77.196, -1.153, 56.66, -22.849, -0.645]
  MoveL 588 to (-16.96, 123.93, 84.62) mm, rotated rx -124.14 ry 0 rz -173.35 deg; joints [9.452, -48.364, 77.108, -1.158, 56.66, -22.569, -0.567]
  MoveL 589 to (-16.68, 124.61, 83.67) mm, rotated rx -124.14 ry 0 rz -173.35 deg; joints [9.417, -48.333, 77.07, -1.159, 56.649, -22.604, -0.549]
  MoveL 590 to (-15.89, 125.18, 82.97) mm, rotated rx -124.14 ry 0 rz -173.35 deg; joints [9.391, -48.292, 77.054, -1.159, 56.614, -22.63, -0.539]
  MoveL 591 to (-15.74, 125.26, 82.89) mm, rotated rx -124.1 ry 0 rz -173.42 deg; joints [9.384, -48.289, 77.045, -1.159, 56.613, -22.601, -0.462]
  MoveL 592 to (-14.94, 125.53, 82.63) mm, rotated rx -124.1 ry 0 rz -173.42 deg; joints [9.373, -48.253, 77.045, -1.157, 56.584, -22.612, -0.468]
  MoveL 593 to (-11.91, 126.15, 82.16) mm, rotated rx -123.81 ry 0 rz -175.1 deg; joints [9.32, -48.265, 76.986, -1.168, 56.583, -22.371, 1.283]
  MoveL 594 to (-8.8, 127.24, 80.87) mm, rotated rx -123.23 ry 0 rz -176.54 deg; joints [9.198, -48.21, 76.845, -1.175, 56.583, -21.911, 2.801]
  MoveL 595 to (-8.25, 127.38, 80.71) mm, rotated rx -123.23 ry 0 rz -176.54 deg; joints [9.191, -48.185, 76.845, -1.174, 56.565, -21.918, 2.796]
  MoveL 596 to (-8.04, 127.41, 80.67) mm, rotated rx -123.22 ry 0 rz -176.63 deg; joints [9.188, -48.184, 76.84, -1.174, 56.565, -21.904, 2.893]
  MoveL 597 to (-7.82, 127.45, 80.64) mm, rotated rx -123.22 ry 0 rz -176.63 deg; joints [9.186, -48.173, 76.84, -1.173, 56.56, -21.906, 2.888]
  MoveL 598 to (-6.62, 127.59, 80.51) mm, rotated rx -123.16 ry 0 rz -177.17 deg; joints [9.174, -48.168, 76.827, -1.173, 56.56, -21.86, 3.438]
  MoveL 599 to (-6.62, 127.59, 80.53) mm, rotated rx -122.88 ry 0 rz -177.84 deg; joints [9.142, -48.239, 76.797, -1.193, 56.56, -21.607, 4.208]
  MoveL 600 to (-4.42, 128.9, 78.57) mm, rotated rx -122.01 ry 0 rz -178.84 deg; joints [8.957, -48.16, 76.591, -1.201, 56.56, -20.916, 5.331]
  MoveL 601 to (-3.96, 129.11, 78.25) mm, rotated rx -122.01 ry 0 rz -178.84 deg; joints [8.945, -48.143, 76.59, -1.202, 56.534, -20.926, 5.341]
  MoveL 602 to (-3.78, 129.17, 78.15) mm, rotated rx -121.96 ry 0 rz -178.92 deg; joints [8.935, -48.139, 76.579, -1.203, 56.534, -20.89, 5.432]
  MoveL 603 to (-3.52, 129.26, 78.02) mm, rotated rx -121.96 ry 0 rz -178.92 deg; joints [8.931, -48.129, 76.579, -1.203, 56.522, -20.894, 5.434]
  MoveL 604 to (-1.85, 129.7, 77.34) mm, rotated rx -121.66 ry 0 rz -179.66 deg; joints [8.866, -48.103, 76.51, -1.205, 56.522, -20.657, 6.213]
  MoveL 605 to (-1.88, 129.69, 77.35) mm, rotated rx -121.39 ry 0 rz 180 deg; joints [8.833, -48.135, 76.478, -1.215, 56.522, -20.412, 6.619]
  MoveL 606 to (0.05, 130.9, 75.32) mm, rotated rx -120.52 ry 0 rz 179.13 deg; joints [8.644, -48.063, 76.281, -1.221, 56.522, -19.728, 7.611]
  MoveL 607 to (2.04, 131.33, 74.53) mm, rotated rx -119.6 ry 0 rz 178.02 deg; joints [8.496, -48.04, 76.135, -1.23, 56.522, -18.958, 8.844]
  MoveL 608 to (2.19, 133.01, 71.49) mm, rotated rx -118.28 ry 0 rz 177.98 deg; joints [8.21, -47.937, 75.857, -1.233, 56.522, -17.923, 9.057]
  MoveL 609 to (2.5, 133.53, 70.5) mm, rotated rx -118.28 ry 0 rz 177.98 deg; joints [8.177, -47.937, 75.852, -1.241, 56.471, -17.952, 9.113]
  MoveL 610 to (3.29, 133.91, 69.74) mm, rotated rx -118.28 ry 0 rz 177.98 deg; joints [8.15, -47.914, 75.852, -1.245, 56.416, -17.976, 9.144]
  MoveL 611 to (3.86, 134.08, 69.39) mm, rotated rx -118.13 ry 0 rz 177.74 deg; joints [8.117, -47.903, 75.822, -1.245, 56.416, -17.859, 9.406]
  MoveL 612 to (4.1, 134.14, 69.26) mm, rotated rx -118.13 ry 0 rz 177.74 deg; joints [8.112, -47.893, 75.822, -1.245, 56.405, -17.864, 9.408]
  MoveL 613 to (10, 135.24, 66.47) mm, rotated rx -116.95 ry 0 rz 175.27 deg; joints [7.855, -47.816, 75.597, -1.245, 56.393, -16.941, 12.029]
  MoveL 614 to (10.53, 135.3, 66.25) mm, rotated rx -116.88 ry 0 rz 175.1 deg; joints [7.838, -47.807, 75.585, -1.245, 56.386, -16.888, 12.209]
  MoveL 615 to (10.74, 135.32, 66.18) mm, rotated rx -116.88 ry 0 rz 175.1 deg; joints [7.835, -47.798, 75.585, -1.244, 56.379, -16.891, 12.207]
  MoveL 616 to (14.37, 135.54, 65.03) mm, rotated rx -116.29 ry 0 rz 173.35 deg; joints [7.715, -47.795, 75.487, -1.248, 56.379, -16.416, 14.059]
  MoveL 617 to (17.64, 136.09, 63.05) mm, rotated rx -115.46 ry 0 rz 172.02 deg; joints [7.534, -47.754, 75.35, -1.248, 56.356, -15.771, 15.501]
  MoveL 618 to (17.92, 136.12, 62.91) mm, rotated rx -115.46 ry 0 rz 172.02 deg; joints [7.529, -47.743, 75.35, -1.247, 56.344, -15.776, 15.502]
  MoveL 619 to (18.45, 136.16, 62.66) mm, rotated rx -115.36 ry 0 rz 171.81 deg; joints [7.507, -47.739, 75.334, -1.247, 56.341, -15.698, 15.731]
  MoveL 620 to (18.4, 136.15, 62.7) mm, rotated rx -115.14 ry 0 rz 171.51 deg; joints [7.481, -47.776, 75.319, -1.254, 56.341, -15.506, 16.085]
  MoveL 621 to (23.58, 137.65, 57.46) mm, rotated rx -112.98 ry 0 rz 169.5 deg; joints [7.005, -47.711, 75.019, -1.254, 56.234, -13.823, 18.427]
  MoveL 622 to (23.57, 137.63, 57.51) mm, rotated rx -112.16 ry 0 rz 169.29 deg; joints [6.893, -47.715, 74.945, -1.252, 56.234, -13.109, 18.714]
  MoveL 623 to (23.29, 138.27, 56.09) mm, rotated rx -111.57 ry 0 rz 169.45 deg; joints [6.764, -47.71, 74.882, -1.252, 56.191, -12.654, 18.655]
  MoveL 624 to (23.25, 138.42, 55.74) mm, rotated rx -111.57 ry 0 rz 169.45 deg; joints [6.752, -47.711, 74.874, -1.252, 56.191, -12.666, 18.664]
  MoveL 625 to (23.25, 138.49, 55.57) mm, rotated rx -111.5 ry 0 rz 169.46 deg; joints [6.737, -47.711, 74.867, -1.252, 56.185, -12.614, 18.669]
  MoveL 626 to (23.25, 138.58, 55.33) mm, rotated rx -111.5 ry 0 rz 169.46 deg; joints [6.729, -47.711, 74.863, -1.252, 56.183, -12.622, 18.675]
  MoveL 627 to (23.37, 139.11, 53.93) mm, rotated rx -110.94 ry 0 rz 169.45 deg; joints [6.603, -47.71, 74.809, -1.252, 56.137, -12.18, 18.781]
  MoveL 628 to (23.32, 139.35, 53.34) mm, rotated rx -110.71 ry 0 rz 169.48 deg; joints [6.552, -47.71, 74.787, -1.252, 56.118, -12.004, 18.786]
  MoveL 629 to (23.65, 140.64, 49.68) mm, rotated rx -109.23 ry 0 rz 169.45 deg; joints [6.223, -47.71, 74.654, -1.245, 56.006, -10.858, 19.062]
  MoveL 630 to (24.07, 140.97, 48.53) mm, rotated rx -109.23 ry 0 rz 169.45 deg; joints [6.184, -47.708, 74.654, -1.246, 55.962, -10.896, 19.103]
  MoveL 631 to (24.75, 141.09, 47.85) mm, rotated rx -109.23 ry 0 rz 169.45 deg; joints [6.16, -47.685, 74.654, -1.245, 55.929, -10.919, 19.113]
  MoveL 632 to (25.64, 141.06, 47.45) mm, rotated rx -109.23 ry 0 rz 169.45 deg; joints [6.146, -47.647, 74.654, -1.242, 55.9, -10.935, 19.103]
  MoveL 633 to (26.99, 140.8, 47.48) mm, rotated rx -109.23 ry 0 rz 169.45 deg; joints [6.145, -47.578, 74.654, -1.234, 55.877, -10.939, 19.058]
  MoveL 634 to (27.66, 140.6, 47.69) mm, rotated rx -109.31 ry 0 rz 169.17 deg; joints [6.163, -47.578, 74.661, -1.235, 55.883, -11.003, 19.325]
  MoveL 635 to (33.53, 138.59, 49.77) mm, rotated rx -110.14 ry 0 rz 166.74 deg; joints [6.348, -47.578, 74.738, -1.241, 55.933, -11.637, 21.629]
  MoveL 636 to (34.49, 138.1, 50.45) mm, rotated rx -110.14 ry 0 rz 166.74 deg; joints [6.369, -47.521, 74.742, -1.234, 55.933, -11.619, 21.568]
  MoveL 637 to (34.94, 137.59, 51.53) mm, rotated rx -110.14 ry 0 rz 166.74 deg; joints [6.404, -47.495, 74.758, -1.232, 55.933, -11.584, 21.526]
  MoveL 638 to (34.99, 137.43, 51.91) mm, rotated rx -110.29 ry 0 rz 166.71 deg; joints [6.439, -47.495, 74.772, -1.233, 55.945, -11.704, 21.532]
  MoveL 639 to (34.9, 137.09, 52.87) mm, rotated rx -110.29 ry 0 rz 166.71 deg; joints [6.472, -47.495, 74.785, -1.233, 55.958, -11.671, 21.507]
  MoveL 640 to (34.24, 136.43, 54.94) mm, rotated rx -111.13 ry 0 rz 166.91 deg; joints [6.658, -47.495, 74.865, -1.234, 56.027, -12.326, 21.16]
  MoveL 641 to (34.22, 136.45, 54.91) mm, rotated rx -112.01 ry 0 rz 166.63 deg; joints [6.778, -47.52, 74.907, -1.233, 56.102, -13.082, 21.35]
  MoveL 642 to (35.06, 135.89, 55.75) mm, rotated rx -112.35 ry 0 rz 166.24 deg; joints [6.854, -47.523, 74.945, -1.233, 56.126, -13.348, 21.676]
  MoveL 643 to (35.03, 135.9, 55.76) mm, rotated rx -112.58 ry 0 rz 165.28 deg; joints [6.889, -47.628, 74.945, -1.242, 56.202, -13.544, 22.667]
  MoveL 644 to (36.59, 135.66, 55.37) mm, rotated rx -112.43 ry 0 rz 164.64 deg; joints [6.854, -47.625, 74.927, -1.242, 56.191, -13.421, 23.332]
  MoveL 645 to (37.62, 135.39, 55.32) mm, rotated rx -112.43 ry 0 rz 164.64 deg; joints [6.851, -47.573, 74.927, -1.236, 56.172, -13.427, 23.299]
  MoveL 646 to (37.97, 135.27, 55.38) mm, rotated rx -112.45 ry 0 rz 164.49 deg; joints [6.856, -47.573, 74.929, -1.236, 56.174, -13.445, 23.446]
  MoveL 647 to (38.54, 135.04, 55.55) mm, rotated rx -112.45 ry 0 rz 164.49 deg; joints [6.861, -47.54, 74.929, -1.231, 56.171, -13.442, 23.415]
  MoveL 648 to (41.47, 133.6, 56.89) mm, rotated rx -113 ry 0 rz 163.18 deg; joints [6.982, -47.549, 74.994, -1.231, 56.206, -13.869, 24.639]
  MoveL 649 to (41.44, 133.61, 56.9) mm, rotated rx -113.08 ry 0 rz 162.74 deg; joints [6.995, -47.599, 74.994, -1.236, 56.237, -13.938, 25.099]
  MoveL 650 to (46.56, 131.98, 56.74) mm, rotated rx -113.02 ry 0 rz 160.53 deg; joints [6.981, -47.598, 74.987, -1.236, 56.233, -13.889, 27.311]
  MoveL 651 to (46.55, 131.99, 56.74) mm, rotated rx -112.91 ry 0 rz 160.1 deg; joints [6.968, -47.659, 74.987, -1.245, 56.233, -13.79, 27.808]
  MoveL 652 to (46.74, 131.96, 56.65) mm, rotated rx -112.87 ry 0 rz 160.02 deg; joints [6.96, -47.658, 74.982, -1.245, 56.231, -13.761, 27.892]
  MoveL 653 to (52.44, 130.85, 54.2) mm, rotated rx -111.89 ry 0 rz 157.74 deg; joints [6.742, -47.644, 74.874, -1.245, 56.156, -12.999, 30.343]
  MoveL 654 to (53.71, 130.41, 54) mm, rotated rx -111.89 ry 0 rz 157.74 deg; joints [6.733, -47.58, 74.875, -1.239, 56.125, -13.011, 30.31]
  MoveL 655 to (54, 130.27, 54.04) mm, rotated rx -111.91 ry 0 rz 157.6 deg; joints [6.736, -47.581, 74.876, -1.239, 56.126, -13.022, 30.439]
  MoveL 656 to (54.41, 130.06, 54.13) mm, rotated rx -111.91 ry 0 rz 157.6 deg; joints [6.738, -47.556, 74.876, -1.236, 56.122, -13.021, 30.419]
  MoveL 657 to (56.76, 128.71, 54.94) mm, rotated rx -112.27 ry 0 rz 156.38 deg; joints [6.815, -47.569, 74.908, -1.236, 56.163, -13.302, 31.583]
  MoveL 658 to (57.14, 128.52, 55.01) mm, rotated rx -112.29 ry 0 rz 156.21 deg; joints [6.822, -47.569, 74.911, -1.236, 56.165, -13.325, 31.752]
  MoveL 659 to (60.62, 126.74, 55.41) mm, rotated rx -112.47 ry 0 rz 154.32 deg; joints [6.86, -47.594, 74.917, -1.235, 56.21, -13.461, 33.608]
